// TwinCAT 3 PLC project Clara_20230328
// ProgramVersion: 3.1.4022.7
// CompilerDefines: VISU_USEWSTRING
// libraries:
//   CAA Memory, * (CAA Technical Workgroup)
//   CmpBitmapPool, * (System)
//   Tc2_EtherCAT, * (Beckhoff Automation GmbH)
//   Tc2_IoFunctions, * (Beckhoff Automation GmbH)
//   Tc2_MC2, * (Beckhoff Automation GmbH)
//   Tc2_MDP, * (Beckhoff Automation GmbH)
//   Tc2_ModbusRTU, * (Beckhoff Automation GmbH)
//   Tc2_SerialCom, * (Beckhoff Automation GmbH)
//   Tc2_Standard, * (Beckhoff Automation GmbH)
//   Tc2_SUPS, * (Beckhoff Automation GmbH)
//   Tc2_System, * (Beckhoff Automation GmbH)
//   Tc2_SystemCX, * (Beckhoff Automation GmbH)
//   Tc2_Utilities, * (Beckhoff Automation GmbH)
//   Tc3_Module, * (Beckhoff Automation GmbH)
//   VisuDialogs, * (System)
//   VisuSymbols,3.5.10.0,System
// project tree:
//   DUTs/01_ST_IO/ ST_Input.TcDUT (not stored), ST_IO_FootPedal.TcDUT (not stored), ST_Output.TcDUT
//   DUTs/02_PLC/ stAxis.TcDUT (not stored), stFootPedal.TcDUT, stISS.TcDUT (not stored), stSubTank.TcDUT (not stored), stMaintenanceUnit.TcDUT, stRollToRoll.TcDUT, stRtu.TcDUT (not stored), stSafetyGuard.TcDUT, stSpitUnit.TcDUT (not stored), stSystemEnvironment.TcDUT, stTableVacuum.TcDUT (not stored), stUpDownSlot.TcDUT, stUVLed.TcDUT (not stored)
//   Enum_Text/Enum/PLC/ AxisStateEnum.TcDUT (not stored), Axis_XY_ErrorEnum.TcDUT (not stored), Axis_Z_ErrorEnum.TcDUT, EnvironmentErrorEnum.TcDUT, EnvironmentStateEnum.TcDUT, FootPedalErrorEnum.TcDUT (not stored), FootPedalStateEnum.TcDUT (not stored), ISSErrorEnum.TcDUT (not stored), SubTankErrorEnum.TcDUT, ISSStateEnum.TcDUT, SubTankInkEnum.TcDUT (not stored), SubTankStateEnum.TcDUT (not stored), MUErrorEnum.TcDUT (not stored), MUStateEnum.TcDUT (not stored), RTRErrorEnum.TcDUT, RTRStateEnum.TcDUT, SafetyGuardErrorEnum.TcDUT, SafetyGuardStateEnum.TcDUT, SpitUnitErrorEnum.TcDUT, SpitUnitStateEnum.TcDUT, SwapInfoEnum.TcDUT (not stored), TabVacErrorEnum.TcDUT, TabVacStateEnum.TcDUT (not stored), UpDownSlotErrorEnum.TcDUT, UpDownSlotStateEnum.TcDUT, UVLedErrorEnum.TcDUT, UVLedStateEnum.TcDUT
//   Enum_Text/Enum/TwinSafe/ TwinSAFE_FB_ESTOP_State_Enum.TcDUT (not stored), TwinSAFE_Group_State_Enum.TcDUT
//   Global Variables/ _01_Global_Variables.TcGVL (not stored), _04_Global_Variables_InOutput.TcGVL (not stored)
//   / GlobalTextList.TcGTLO (not stored), ImagePool.TcIPO (not stored), PlcTask.TcTTO (not stored), Task_com.TcTTO (not stored), 视图管理器.TcVMO (not stored)
//   GVLs/ COMM.TcGVL (not stored), GVL.TcGVL (not stored), GVL_Alarm.TcGVL (not stored), GVL_API.TcGVL
//   POUs/000_程序辅助系统/报警/Data types/ Alm_AlarmHistoryType.TcDUT, Alm_AlarmType.TcDUT (not stored), Alm_AlmMsg.TcDUT (not stored), Alm_EventClass.TcDUT (not stored)
//   POUs/000_程序辅助系统/报警/diag_FB/ ethercatinfo_read.TcPOU
//   POUs/000_程序辅助系统/报警/Alarm_FB/ FB_AlarmMain.TcPOU (not stored), FB_DiagDataLogging_S.TcPOU, FB_SetAlarm.TcPOU, SW_FormatWstring.TcPOU (not stored)
//   POUs/000_程序辅助系统/报警/Alarm_FB/Products/ FB_DirectoryCopy.TcPOU, FB_FileCopy.TcPOU (not stored)
//   POUs/000_程序辅助系统/报警/ MAIN_Alarm.TcPOU
//   POUs/000_程序辅助系统/系统功能/ P_UPS.TcPOU, systime.TcPOU (not stored)
//   POUs/001_FB/ FB_Buzzer.TcPOU (not stored), FB_count.TcPOU, FB_SQUARE.TcPOU (not stored), FB_WriteAnalog.TcPOU
//   POUs/002_Modbus/BackPrg/ PRG_COMM.TcPOU (not stored)
//   POUs/002_Modbus/ PRG_SerialComm.TcPOU, P_Modbus.TcPOU (not stored), P_Modbus_RTU.TcPOU
//   POUs/003_Input_Output/ IO_Link.TcPOU (not stored), P_API_IO.TcPOU
//   POUs/010_Motion/MotionBase/ FB_Home_Z.TcPOU, FB_Home_X.TcPOU (not stored), FB_MoveFS_Exte.TcPOU (not stored), FB_MoveSS_Exte.TcPOU (not stored), FB_MoveZ_Exte.TcPOU (not stored)
//   POUs/010_Motion/XMove/ P_FastScan.TcPOU (not stored)
//   POUs/010_Motion/YMove/ P_SlowScan.TcPOU (not stored)
//   POUs/010_Motion/ZMove/ P_Z_Axis.TcPOU (not stored)
//   POUs/030_MediaTransport/TableVacuum/FB/ FB_TableVacuum.TcPOU
//   POUs/030_MediaTransport/UpDownSlot/FB/ FB_UpDownSlotS1.TcPOU (not stored), FB_UpDownSlotS2_S6.TcPOU (not stored)
//   POUs/040_System/FootPedal/FB/ FB_FootPedal.TcPOU (not stored)
//   POUs/040_System/SafetyGuard/FB/ FB_SafetyGuard.TcPOU
//   POUs/040_System/SafetyGuard/ P_SafetyGuard.TcPOU
//   POUs/040_System/SystemEnvironment/FB/ FB_SystemEnvironment.TcPOU (not stored)
//   POUs/050_InkSystem/ISS/ P_ISS.TcPOU (not stored)
//   POUs/050_InkSystem/ P_InkSystem.TcPOU
//   POUs/050_InkSystem/搅拌_吸废墨/FB/ FB_Stirrer.TcPOU
//   POUs/050_InkSystem/搅拌_吸废墨/ P_Stirrer_WastePump.TcPOU
//   POUs/030_MediaTransport/ P_MediaTransport.TcPOU (not stored)
//   POUs/030_MediaTransport/TableVacuum/ P_TableVacuum.TcPOU
//   POUs/030_MediaTransport/UpDownSlot/ P_UpDownSlot.TcPOU
//   POUs/010_Motion/MotionBase/PTP/ Axis_IO.TcPOU (not stored), Axis_PTP_CoE.TcPOU
//   POUs/010_Motion/ P_Motion.TcPOU
//   POUs/060_UVLed/FB/ FB_UVLed_L.TcPOU, FB_UVLed_R.TcPOU
//   POUs/070_RollToRoll/FB/ FB_RollToRoll_Torque.TcPOU (not stored)
//   POUs/100_SubTank/FB/ FB_Circulation.TcPOU (not stored), FB_SubTank_C.TcPOU (not stored), FB_SubTank_W.TcPOU (not stored)
//   POUs/100_SubTank/ P_SubTank.TcPOU
//   POUs/999_TwinSAFE/ P_TwinSAFE.TcPOU (not stored)
//   POUs/ MAIN.TcPOU
//   POUs/070_RollToRoll/ P_RollToRoll.TcPOU
//   POUs/040_System/FootPedal/ P_FootPedal.TcPOU
//   POUs/040_System/ P_System.TcPOU
//   POUs/040_System/SystemEnvironment/ P_SystemEnvironment.TcPOU (not stored)
//   POUs/060_UVLed/ P_UVLed.TcPOU
//   POUs/090MaintenanceUnit/FB/ FB_Auto_Cycles_Swap.TcPOU, FB_drip_purge.TcPOU (not stored)
//   POUs/090MaintenanceUnit/ P_MaintenanceUnit.TcPOU
//   POUs/080SpitUnit/FB/ FB_HomeSpitUnit.TcPOU (not stored), FB_MoveSpitUnit_Exte.TcPOU (not stored)
//   POUs/080SpitUnit/ P_SpitUnit.TcPOU (not stored)
//   VISUs/base/ title.TcVIS (not stored)
//   VISUs/Components/IO_Components/ F99_IO_IO.TcVIS (not stored), F99_IO_IO_1.TcVIS (not stored), F99_IO_IO_2.TcVIS (not stored)
//   VISUs/Components/ VIS_FootPedal.TcVIS, VIS_Drip_purge.TcVIS, VIS_SubTank.TcVIS (not stored), VIS_SystemEnvironment.TcVIS, VIS_ISS.TcVIS, VIS_MU.TcVIS, VIS_RTR_1.TcVIS, VIS_RTR_2.TcVIS (not stored), VIS_SaftyGuard.TcVIS, VIS_SpitUnit.TcVIS (not stored), VIS_TabVac.TcVIS (not stored), VIS_UpDownSlot.TcVIS (not stored)
//   VISUs/HMI_IO监控文字/ EL1809_M_1.TcTLO (not stored), EL1809_M_2.TcTLO (not stored), EL1809_M_3.TcTLO (not stored), EL1809_S_1.TcTLO (not stored), EL1809_S_2.TcTLO, EL1904_M_1.TcTLO (not stored), EL1904_M_2.TcTLO (not stored), EL1904_M_3.TcTLO, EL1904_M_4.TcTLO, EL1904_M_5.TcTLO, EL2809_M_1.TcTLO, EL2809_M_2.TcTLO, EL2809_M_3.TcTLO, EL2809_M_4.TcTLO (not stored), EL2809_S_1.TcTLO, EL2904_M_1.TcTLO
//   VISUs/ F99_Monitor.TcVIS, F7_RTR.TcVIS (not stored), F4_System.TcVIS, F1_AXIS.TcVIS (not stored), F5_InkSystem.TcVIS (not stored), F3_MediaTransport.TcVIS, F6_UVLed.TcVIS
//   VISUs/VIS文本/PLC/ ISS_Object.TcTLO (not stored), subinklevel.TcTLO, TextListSpitUnitErrorid.TcTLO, TextListSpitUnitState.TcTLO (not stored), TextList_EnvironmentError.TcTLO (not stored), TextList_EnvironmentState.TcTLO (not stored), TextList_FootPedalerroid.TcTLO, TextList_SubTankerroid.TcTLO (not stored), TextList_FootPedalstate.TcTLO (not stored), TextList_ISSerrorid.TcTLO (not stored), TextList_ISSstate.TcTLO (not stored), TextList_MU_errorid.TcTLO (not stored), TextList_MU_state.TcTLO (not stored), TextList_RTRstate.TcTLO, TextList_RTR_errorid.TcTLO (not stored), TextList_SafetyGuarderrorid.TcTLO, TextList_SafetyGuardstate.TcTLO (not stored), TextList_SubTank_circuit.TcTLO (not stored), TextList_SwapInfo.TcTLO (not stored), TextList_tabvac_errorid.TcTLO (not stored), TextList_tabvac_state.TcTLO (not stored), TextList_UpDownSlot_errorid.TcTLO (not stored), TextList_UpDownSlot_state.TcTLO (not stored), TextList_UVLed_errorid.TcTLO, TextList_UVLed_state.TcTLO, TextList_xyErrorid.TcTLO (not stored), TextList_xyzState.TcTLO (not stored), TextList_zErrorid.TcTLO
//   VISUs/VIS文本/TwinSafe/ TextList_TwinSAFE_FB_ESTOP_State.TcTLO (not stored), TextList_TwinSAFE_Group_State.TcTLO (not stored)
//   VISUs/报警/ Visualization_ActEvent.TcVIS (not stored), Visualization_LogEvent.TcVIS, vis_arm.TcVIS (not stored)
// real-time tasks:
//   TASK PlcTask: cycle T#10ms, priority 12, ADS port 350
//   TASK Task_com: cycle T#2ms, priority 6, ADS port 352
// motion (NC):
//   TASK NC-Task 1 SAF: cycle T#2ms, priority 4, ADS port 501
//   TASK NC-Task 1 SVB: cycle T#5ms, priority 10, ADS port 511
//   AXIS Axis_FS (id 1)
//     Dynamic: Acceleration=5927.27, Deceleration=5927.27, Jerk=27883
//     Velo: RefSearch=10, RefSync=10, SlowManual=50, FastManual=100
//     TargetPosControl: Time=0.005
//     OtherSettings: AllowMotionCmdToSlave=true
//     encoder EncType=19
//       EncPara: ScaleFactorNumerator=0.001, MaxCount=#xffffffff
//         Inc: RefSearchInverse=true, RefSyncInverse=false
//     drive DrvType=16
//       DrvPara: MaxCount=#xffffffff, DriveControlDWord=#x00020000
//         Analog: VeloReferenz=2000, TorqueSetpointScale=10, ScaleFactorActTorque=0.1
//         TimeComp: TaskDelayCycles=1
//     controller CtrType=1
//       CtrPara: PriorControlFactor=1
//         PosDiffControl: Range=250
//         Observer: BandWidth=20
//   AXIS Axis_SS (id 2)
//     Dynamic: Acceleration=274.92, Deceleration=274.92, Jerk=748.92
//     Velo: Maximum=174
//     OtherSettings: AllowMotionCmdToSlave=true
//     encoder EncType=19
//       EncPara: ScaleFactorNumerator=3.12605035e-07, Inverse=true, MaxCount=#xffffffff
//     drive DrvType=16
//       DrvPara: Inverse=true, MaxCount=#xffffffff, DriveControlDWord=#x00020000
//         Analog: VeloReferenz=180, TorqueSetpointScale=10, ScaleFactorActTorque=0.1
//         TimeComp: TaskDelayCycles=1
//     controller CtrType=1
//       CtrPara: PriorControlFactor=1
//         PosDiffControl: Range=50
//         Observer: BandWidth=20
//   AXIS Z_Axis (id 3)
//     Dynamic: Acceleration=33.4286, Deceleration=33.4286, Jerk=133.032
//     Velo: RefSearch=2, RefSync=2, SlowManual=8, FastManual=10, Maximum=15
//     OtherSettings: AllowMotionCmdToSlave=true
//     encoder EncType=19
//       EncPara: ScaleFactorNumerator=1.7881393e-08, MaxCount=#xffffffff
//         Inc: RefSearchInverse=true, RefSyncInverse=false
//     drive DrvType=16
//       DrvPara: MaxCount=#xffffffff, DriveControlDWord=#x00020000
//         Analog: VeloReferenz=15, TorqueSetpointScale=10, ScaleFactorActTorque=0.1
//         TimeComp: TaskDelayCycles=1
//     controller CtrType=1
//       CtrPara: PriorControlFactor=1
//         PosDiffControl: Range=10
//         Observer: BandWidth=20
//   AXIS Axis_unwider_input1 (id 4)
//     Dynamic: Acceleration=4200, Deceleration=4200, Jerk=14700
//     Velo: SlowManual=60, FastManual=100, Maximum=3000
//     OtherSettings: AllowMotionCmdToSlave=true
//     encoder EncType=19
//       EncPara: ScaleFactorNumerator=3.57628e-06, MaxCount=#xffffffff
//     drive DrvType=16
//       DrvPara: MaxCount=#xffffffff, DriveControlDWord=#x00020000
//         Analog: VeloReferenz=3000, TorqueSetpointScale=10, ScaleFactorActTorque=0.1
//         TimeComp: TaskDelayCycles=1
//     controller CtrType=1
//       CtrPara: PriorControlFactor=1
//         PosDiffControl: Enable=false, Range=100
//         Observer: BandWidth=20
//   AXIS Axis_unwinder_input2 (id 5)
//     Dynamic: Acceleration=4000, Deceleration=4000, Jerk=16000
//     Velo: Maximum=3000
//     OtherSettings: AllowMotionCmdToSlave=true
//     encoder EncType=19
//       EncPara: ScaleFactorNumerator=3.57628e-06, Inverse=true, MaxCount=#xffffffff
//     drive DrvType=16
//       DrvPara: Inverse=true, MaxCount=#xffffffff, DriveControlDWord=#x00020000
//         Analog: VeloReferenz=3000, TorqueSetpointScale=10, ScaleFactorActTorque=0.1
//         TimeComp: TaskDelayCycles=1
//     controller CtrType=1
//       CtrPara: PriorControlFactor=1
//         PosDiffControl: Enable=false, Range=100
//         Observer: BandWidth=20
//   AXIS Axis_winder_output1 (id 6)
//     Dynamic: Acceleration=4000, Deceleration=4000, Jerk=16000
//     Velo: Maximum=3000
//     OtherSettings: AllowMotionCmdToSlave=true
//     encoder EncType=19
//       EncPara: ScaleFactorNumerator=3.57628e-06, MaxCount=#xffffffff
//     drive DrvType=16
//       DrvPara: MaxCount=#xffffffff, DriveControlDWord=#x00020000
//         Analog: VeloReferenz=3000, TorqueSetpointScale=10, ScaleFactorActTorque=0.1
//         TimeComp: TaskDelayCycles=1
//     controller CtrType=1
//       CtrPara: PriorControlFactor=1
//         PosDiffControl: Enable=false, Range=100
//         Observer: BandWidth=20
//   AXIS Axis_winder_output2 (id 7)
//     Dynamic: Acceleration=4000, Deceleration=4000, Jerk=16000
//     Velo: Maximum=3000
//     OtherSettings: AllowMotionCmdToSlave=true
//     encoder EncType=19
//       EncPara: ScaleFactorNumerator=3.57628e-06, Inverse=true, MaxCount=#xffffffff
//     drive DrvType=16
//       DrvPara: Inverse=true, MaxCount=#xffffffff, DriveControlDWord=#x00020000
//         Analog: VeloReferenz=3000, TorqueSetpointScale=10, ScaleFactorActTorque=0.1
//         TimeComp: TaskDelayCycles=1
//     controller CtrType=1
//       CtrPara: PriorControlFactor=1
//         PosDiffControl: Enable=false, Range=100
//         Observer: BandWidth=20
//   AXIS SpitUnit (id 8)
//     Dynamic: Acceleration=32.1429, Deceleration=32.1429, Jerk=137.755
//     Velo: RefSearch=2, RefSync=2, SlowManual=5, FastManual=10, Maximum=15
//     OtherSettings: AllowMotionCmdToSlave=true
//     encoder EncType=19
//       EncPara: ScaleFactorNumerator=1.7881393e-08, Inverse=true, MaxCount=#xffffffff
//         Inc: RefSearchInverse=true, RefSyncInverse=false
//     drive DrvType=16
//       DrvPara: Inverse=true, MaxCount=#xffffffff, DriveControlDWord=#x00020000
//         Analog: VeloReferenz=15, TorqueSetpointScale=10, ScaleFactorActTorque=0.1
//         TimeComp: TaskDelayCycles=1
//     controller CtrType=1
//       CtrPara: PriorControlFactor=1
//         PosDiffControl: Range=10
//         Observer: BandWidth=20
// I/O:
//   DEVICE Device 1 (EtherCAT), AmsNetId 192.168.1.138.2.1
//     Term 1 (EK1200) [EK1200-5000 EtherCAT Power supply (2A E-Bus)]
//       Term 2 (EL1809) [EL1809 16Ch. Dig. Input 24V, 3ms]
//       Term 3 (EL1809) [EL1809 16Ch. Dig. Input 24V, 3ms]
//       Term 4 (EL1809) [EL1809 16Ch. Dig. Input 24V, 3ms]
//       Term 5 (EL2809) [EL2809 16Ch. Dig. Output 24V, 0.5A]
//       Term 6 (EL2809) [EL2809 16Ch. Dig. Output 24V, 0.5A]
//       Term 7 (EL2809) [EL2809 16Ch. Dig. Output 24V, 0.5A]
//       Term 8 (EL6900) [EL6900, TwinSAFE PLC]
//       Term 9 (EL1904) [EL1904, 4 Ch. Safety Input 24V, TwinSAFE]
//         modules: Module 1 (FSOES)
//       Term 10 (EL1904) [EL1904, 4 Ch. Safety Input 24V, TwinSAFE]
//         modules: Module 1 (FSOES)
//       Term 11 (EL1904) [EL1904, 4 Ch. Safety Input 24V, TwinSAFE]
//         modules: Module 1 (FSOES)
//       Term 12 (EL1904) [EL1904, 4 Ch. Safety Input 24V, TwinSAFE]
//         modules: Module 1 (FSOES)
//       Term 13 (EL1904) [EL1904, 4 Ch. Safety Input 24V, TwinSAFE]
//         modules: Module 1 (FSOES)
//       Term 14 (EL9410) [EL9410 E-Bus Power Supplier  (Diagnostics)]
//       Term 15 (EL2904) [EL2904, 4 Ch. Safety Output 24V, 0.5A, TwinSAFE]
//         modules: Module 1 (FSOES), Module 2 (DO)
//       Term 16 (EL2809) [EL2809 16Ch. Dig. Output 24V, 0.5A]
//       Term 17 (EL6001) [EL6001 Interface (RS232)]
//       Term 18 (EL6022) [EL6022 Interface 2Ch. (RS422/485)]
//       Term 19 (EK1110) [EK1110 EtherCAT extension]
//     Drive 20 (ASDA-A3-E CoE Drive) [Delta ASDA-A3-E EtherCAT(CoE) Drive Rev0.05]
//     Drive 21 (ASDA-A3-E CoE Drive) [Delta ASDA-A3-E EtherCAT(CoE) Drive Rev0.05]
//     Drive 22 (ASDA-A3-E CoE Drive) [Delta ASDA-A3-E EtherCAT(CoE) Drive Rev0.05]
//     Drive 23 (ASDA-A3-E CoE Drive) [Delta ASDA-A3-E EtherCAT(CoE) Drive Rev0.05]
//     Drive 24 (ASDA-A3-E CoE Drive) [Delta ASDA-A3-E EtherCAT(CoE) Drive Rev0.05]
//     Drive 25 (ASDA-A3-E CoE Drive) [Delta ASDA-A3-E EtherCAT(CoE) Drive Rev0.05]
//     Drive 26 (ASDA-A3-E CoE Drive) [Delta ASDA-A3-E EtherCAT(CoE) Drive Rev0.05]
//     Drive 27 (ASDA-A3-E CoE Drive) [Delta ASDA-A3-E EtherCAT(CoE) Drive Rev0.05]
//     Term 28 (EK1100) [EK1100 EtherCAT Coupler (2A E-Bus)]
//       Term 29 (EL1809) [EL1809 16Ch. Dig. Input 24V, 3ms]
//       Term 30 (EL1809) [EL1809 16Ch. Dig. Input 24V, 3ms]
//       Term 31 (EL2809) [EL2809 16Ch. Dig. Output 24V, 0.5A]
//       Term 32 (EL4002) [EL4002 2Ch. Ana. Output 0-10V, 12bit]
//       Term 33 (EL9011) [EL9011 End Terminal]
// variable links:
//   Device 1 (EtherCAT) <-> Device 1 (EtherCAT)/Term 1 (EK1200)/Term 10 (EL1904)
//     Term 1 (EK1200)/Term 8 (EL6900)/ConnectionInputs/Message_53 TxPDO <-> Module 1 (FSOES)/RxPDO/FSOE
//   Device 1 (EtherCAT) <-> Device 1 (EtherCAT)/Term 1 (EK1200)/Term 12 (EL1904)
//     Term 1 (EK1200)/Term 8 (EL6900)/ConnectionOutputs/Message_55 RxPDO <-> Module 1 (FSOES)/TxPDO/FSOE
//   Device 1 (EtherCAT) <-> Device 1 (EtherCAT)/Term 1 (EK1200)/Term 13 (EL1904)
//     Term 1 (EK1200)/Term 8 (EL6900)/ConnectionInputs/Message_56 TxPDO <-> Module 1 (FSOES)/RxPDO/FSOE
//     Term 1 (EK1200)/Term 8 (EL6900)/ConnectionOutputs/Message_56 RxPDO <-> Module 1 (FSOES)/TxPDO/FSOE
//   Device 1 (EtherCAT) <-> Device 1 (EtherCAT)/Term 1 (EK1200)/Term 15 (EL2904)
//     Term 1 (EK1200)/Term 8 (EL6900)/ConnectionInputs/Message_57 TxPDO <-> Module 1 (FSOES)/RxPDO/FSOE
//   Device 1 (EtherCAT) <-> Device 1 (EtherCAT)/Term 1 (EK1200)/Term 8 (EL6900)
//     Term 1 (EK1200)/Term 10 (EL1904)/Module 1 (FSOES)/TxPDO/FSOE <-> ConnectionOutputs/Message_53 RxPDO
//     Term 1 (EK1200)/Term 11 (EL1904)/Module 1 (FSOES)/TxPDO/FSOE <-> ConnectionOutputs/Message_58 RxPDO
//     Term 1 (EK1200)/Term 15 (EL2904)/Module 1 (FSOES)/TxPDO/FSOE <-> ConnectionOutputs/Message_57 RxPDO
//     Term 1 (EK1200)/Term 11 (EL1904)/Module 1 (FSOES)/RxPDO/FSOE <-> ConnectionInputs/Message_58 TxPDO
//     Term 1 (EK1200)/Term 12 (EL1904)/Module 1 (FSOES)/RxPDO/FSOE <-> ConnectionInputs/Message_55 TxPDO
//     Term 1 (EK1200)/Term 9 (EL1904)/Module 1 (FSOES)/RxPDO/FSOE <-> ConnectionInputs/Message_52 TxPDO
//   Device 1 (EtherCAT) <-> Device 1 (EtherCAT)/Term 1 (EK1200)/Term 9 (EL1904)
//     Term 1 (EK1200)/Term 8 (EL6900)/ConnectionOutputs/Message_52 RxPDO <-> Module 1 (FSOES)/TxPDO/FSOE
//   NC-Task 1 SAF/Axes/Axis_FS <-> Device 1 (EtherCAT)/Drive 20 (ASDA-A3-E CoE Drive)
//     Drive/Inputs/In/nDataIn3[0] <-> 2nd TxPDO Mapping/Actual Torque
//     Drive/Inputs/In/nDcOutputTime <-> InfoData/DcOutputShift
//     Drive/Inputs/In/nState1 <-> 2nd TxPDO Mapping/Status Word
//     Drive/Inputs/In/nState2 <-> 2nd TxPDO Mapping/Status Word @bit 8
//     Drive/Inputs/In/nState4 @bit 1 <-> WcState/InputToggle
//     Drive/Inputs/In/nState4 <-> WcState/WcState
//     Drive/Outputs/Out/nCtrl1 <-> 2nd RxPDO Mapping/Control Word
//     Drive/Outputs/Out/nCtrl2 <-> 2nd RxPDO Mapping/Control Word @bit 8
//     Drive/Outputs/Out/nDataOut1 <-> 2nd RxPDO Mapping/Target Position
//     Drive/Outputs/Out/nDataOut2 <-> 2nd RxPDO Mapping/Target Velocity
//     Drive/Outputs/Out/nDataOut4[0] <-> 2nd RxPDO Mapping/Target Torque
//     Enc/Inputs/In/nDataIn1 <-> 2nd TxPDO Mapping/Actual Position
//     Enc/Inputs/In/nDataIn3 <-> 2nd TxPDO Mapping/Touch Probe Pos1 Pos Value
//     Enc/Inputs/In/nDataIn7 <-> 2nd TxPDO Mapping/Velocity actual value
//     Enc/Inputs/In/nDcInputTime <-> InfoData/DcInputShift
//     Enc/Inputs/In/nState4 @bit 1 <-> WcState/InputToggle
//     Enc/Inputs/In/nState4 <-> WcState/WcState
//     Enc/Inputs/In/nState5 <-> 2nd TxPDO Mapping/Touch Probe Status
//     Enc/Inputs/In/nState6 <-> 2nd TxPDO Mapping/Touch Probe Status @bit 8
//     Enc/Outputs/Out/nCtrl5 <-> 2nd RxPDO Mapping/Touch Probe Function
//     Enc/Outputs/Out/nCtrl6 <-> 2nd RxPDO Mapping/Touch Probe Function @bit 8
//   NC-Task 1 SAF/Axes/Axis_SS <-> Device 1 (EtherCAT)/Drive 21 (ASDA-A3-E CoE Drive)
//     Drive/Inputs/In/nDataIn3[0] <-> 2nd TxPDO Mapping/Actual Torque
//     Drive/Inputs/In/nDcOutputTime <-> InfoData/DcOutputShift
//     Drive/Inputs/In/nState1 <-> 2nd TxPDO Mapping/Status Word
//     Drive/Inputs/In/nState2 <-> 2nd TxPDO Mapping/Status Word @bit 8
//     Drive/Inputs/In/nState4 @bit 1 <-> WcState/InputToggle
//     Drive/Inputs/In/nState4 <-> WcState/WcState
//     Drive/Outputs/Out/nCtrl1 <-> 2nd RxPDO Mapping/Control Word
//     Drive/Outputs/Out/nCtrl2 <-> 2nd RxPDO Mapping/Control Word @bit 8
//     Drive/Outputs/Out/nDataOut1 <-> 2nd RxPDO Mapping/Target Position
//     Drive/Outputs/Out/nDataOut2 <-> 2nd RxPDO Mapping/Target Velocity
//     Drive/Outputs/Out/nDataOut4[0] <-> 2nd RxPDO Mapping/Target Torque
//     Enc/Inputs/In/nDataIn1 <-> 2nd TxPDO Mapping/Actual Position
//     Enc/Inputs/In/nDataIn3 <-> 2nd TxPDO Mapping/Touch Probe Pos1 Pos Value
//     Enc/Inputs/In/nDataIn7 <-> 2nd TxPDO Mapping/Velocity actual value
//     Enc/Inputs/In/nDcInputTime <-> InfoData/DcInputShift
//     Enc/Inputs/In/nState4 @bit 1 <-> WcState/InputToggle
//     Enc/Inputs/In/nState4 <-> WcState/WcState
//     Enc/Inputs/In/nState5 <-> 2nd TxPDO Mapping/Touch Probe Status
//     Enc/Inputs/In/nState6 <-> 2nd TxPDO Mapping/Touch Probe Status @bit 8
//     Enc/Outputs/Out/nCtrl5 <-> 2nd RxPDO Mapping/Touch Probe Function
//     Enc/Outputs/Out/nCtrl6 <-> 2nd RxPDO Mapping/Touch Probe Function @bit 8
//   NC-Task 1 SAF/Axes/Axis_unwider_input1 <-> Device 1 (EtherCAT)/Drive 23 (ASDA-A3-E CoE Drive)
//     Drive/Inputs/In/nDataIn3[0] <-> 3rd TxPDO Mapping/Actual Torque
//     Drive/Inputs/In/nDcOutputTime <-> InfoData/DcOutputShift
//     Drive/Inputs/In/nState1 <-> 3rd TxPDO Mapping/Status Word
//     Drive/Inputs/In/nState2 <-> 3rd TxPDO Mapping/Status Word @bit 8
//     Drive/Inputs/In/nState4 @bit 1 <-> WcState/InputToggle
//     Drive/Inputs/In/nState4 <-> WcState/WcState
//     Drive/Inputs/In/nState5 <-> 3rd TxPDO Mapping/Mode Of Operation Display
//     Drive/Outputs/Out/nCtrl1 <-> 3rd RxPDO Mapping/Control Word
//     Drive/Outputs/Out/nCtrl2 <-> 3rd RxPDO Mapping/Control Word @bit 8
//     Drive/Outputs/Out/nCtrl5 <-> 3rd RxPDO Mapping/Mode Of Operation
//     Drive/Outputs/Out/nDataOut1 <-> 3rd RxPDO Mapping/Target Position
//     Drive/Outputs/Out/nDataOut2 <-> 3rd RxPDO Mapping/Target Velocity
//     Drive/Outputs/Out/nDataOut4[0] <-> 3rd RxPDO Mapping/Target Torque
//     Enc/Inputs/In/nDataIn1 <-> 3rd TxPDO Mapping/Actual Position
//     Enc/Inputs/In/nDataIn3 <-> 3rd TxPDO Mapping/Touch Probe Pos1 Pos Value
//     Enc/Inputs/In/nDataIn7 <-> 3rd TxPDO Mapping/Velocity actual value
//     Enc/Inputs/In/nDcInputTime <-> InfoData/DcInputShift
//     Enc/Inputs/In/nState4 @bit 1 <-> WcState/InputToggle
//     Enc/Inputs/In/nState4 <-> WcState/WcState
//     Enc/Inputs/In/nState5 <-> 3rd TxPDO Mapping/Touch Probe Status
//     Enc/Inputs/In/nState6 <-> 3rd TxPDO Mapping/Touch Probe Status @bit 8
//     Enc/Outputs/Out/nCtrl5 <-> 3rd RxPDO Mapping/Touch Probe Function
//     Enc/Outputs/Out/nCtrl6 <-> 3rd RxPDO Mapping/Touch Probe Function @bit 8
//   NC-Task 1 SAF/Axes/Axis_unwinder_input2 <-> Device 1 (EtherCAT)/Drive 24 (ASDA-A3-E CoE Drive)
//     Drive/Inputs/In/nDataIn3[0] <-> 3rd TxPDO Mapping/Actual Torque
//     Drive/Inputs/In/nDcOutputTime <-> InfoData/DcOutputShift
//     Drive/Inputs/In/nState1 <-> 3rd TxPDO Mapping/Status Word
//     Drive/Inputs/In/nState2 <-> 3rd TxPDO Mapping/Status Word @bit 8
//     Drive/Inputs/In/nState4 @bit 1 <-> WcState/InputToggle
//     Drive/Inputs/In/nState4 <-> WcState/WcState
//     Drive/Inputs/In/nState5 <-> 3rd TxPDO Mapping/Mode Of Operation Display
//     Drive/Outputs/Out/nCtrl1 <-> 3rd RxPDO Mapping/Control Word
//     Drive/Outputs/Out/nCtrl2 <-> 3rd RxPDO Mapping/Control Word @bit 8
//     Drive/Outputs/Out/nCtrl5 <-> 3rd RxPDO Mapping/Mode Of Operation
//     Drive/Outputs/Out/nDataOut1 <-> 3rd RxPDO Mapping/Target Position
//     Drive/Outputs/Out/nDataOut2 <-> 3rd RxPDO Mapping/Target Velocity
//     Drive/Outputs/Out/nDataOut4[0] <-> 3rd RxPDO Mapping/Target Torque
//     Enc/Inputs/In/nDataIn1 <-> 3rd TxPDO Mapping/Actual Position
//     Enc/Inputs/In/nDataIn3 <-> 3rd TxPDO Mapping/Touch Probe Pos1 Pos Value
//     Enc/Inputs/In/nDataIn7 <-> 3rd TxPDO Mapping/Velocity actual value
//     Enc/Inputs/In/nDcInputTime <-> InfoData/DcInputShift
//     Enc/Inputs/In/nState4 @bit 1 <-> WcState/InputToggle
//     Enc/Inputs/In/nState4 <-> WcState/WcState
//     Enc/Inputs/In/nState5 <-> 3rd TxPDO Mapping/Touch Probe Status
//     Enc/Inputs/In/nState6 <-> 3rd TxPDO Mapping/Touch Probe Status @bit 8
//     Enc/Outputs/Out/nCtrl5 <-> 3rd RxPDO Mapping/Touch Probe Function
//     Enc/Outputs/Out/nCtrl6 <-> 3rd RxPDO Mapping/Touch Probe Function @bit 8
//   NC-Task 1 SAF/Axes/Axis_winder_output1 <-> Device 1 (EtherCAT)/Drive 25 (ASDA-A3-E CoE Drive)
//     Drive/Inputs/In/nDataIn3[0] <-> 3rd Transmit PDO Mapping/Torque actual value
//     Drive/Inputs/In/nDcOutputTime <-> InfoData/DcOutputShift
//     Drive/Inputs/In/nState1 <-> 3rd Transmit PDO Mapping/Statusword
//     Drive/Inputs/In/nState2 <-> 3rd Transmit PDO Mapping/Statusword @bit 8
//     Drive/Inputs/In/nState4 @bit 1 <-> WcState/InputToggle
//     Drive/Inputs/In/nState4 <-> WcState/WcState
//     Drive/Inputs/In/nState5 <-> 3rd Transmit PDO Mapping/Modes of operation display
//     Drive/Outputs/Out/nCtrl1 <-> 3rd Receive PDO Mapping/Controlword
//     Drive/Outputs/Out/nCtrl2 <-> 3rd Receive PDO Mapping/Controlword @bit 8
//     Drive/Outputs/Out/nCtrl5 <-> 3rd Receive PDO Mapping/Modes of operation
//     Drive/Outputs/Out/nDataOut1 <-> 3rd Receive PDO Mapping/Target position
//     Drive/Outputs/Out/nDataOut2 <-> 3rd Receive PDO Mapping/Target velocity
//     Drive/Outputs/Out/nDataOut4[0] <-> 3rd Receive PDO Mapping/Target torque
//     Enc/Inputs/In/nDataIn1 <-> 3rd Transmit PDO Mapping/Position actual value
//     Enc/Inputs/In/nDataIn3 <-> 3rd Transmit PDO Mapping/Touch Probe Pos1 Pos Value
//     Enc/Inputs/In/nDataIn7 <-> 3rd Transmit PDO Mapping/Velocity actual value
//     Enc/Inputs/In/nDcInputTime <-> InfoData/DcInputShift
//     Enc/Inputs/In/nState4 @bit 1 <-> WcState/InputToggle
//     Enc/Inputs/In/nState4 <-> WcState/WcState
//     Enc/Inputs/In/nState5 <-> 3rd Transmit PDO Mapping/Touch Probe Status
//     Enc/Inputs/In/nState6 <-> 3rd Transmit PDO Mapping/Touch Probe Status @bit 8
//     Enc/Outputs/Out/nCtrl5 <-> 3rd Receive PDO Mapping/Touch Probe Function
//     Enc/Outputs/Out/nCtrl6 <-> 3rd Receive PDO Mapping/Touch Probe Function @bit 8
//   NC-Task 1 SAF/Axes/Axis_winder_output2 <-> Device 1 (EtherCAT)/Drive 26 (ASDA-A3-E CoE Drive)
//     Drive/Inputs/In/nDataIn3[0] <-> 3rd TxPDO Mapping/Actual Torque
//     Drive/Inputs/In/nDcOutputTime <-> InfoData/DcOutputShift
//     Drive/Inputs/In/nState1 <-> 3rd TxPDO Mapping/Status Word
//     Drive/Inputs/In/nState2 <-> 3rd TxPDO Mapping/Status Word @bit 8
//     Drive/Inputs/In/nState4 @bit 1 <-> WcState/InputToggle
//     Drive/Inputs/In/nState4 <-> WcState/WcState
//     Drive/Inputs/In/nState5 <-> 3rd TxPDO Mapping/Mode Of Operation Display
//     Drive/Outputs/Out/nCtrl1 <-> 3rd RxPDO Mapping/Control Word
//     Drive/Outputs/Out/nCtrl2 <-> 3rd RxPDO Mapping/Control Word @bit 8
//     Drive/Outputs/Out/nCtrl5 <-> 3rd RxPDO Mapping/Mode Of Operation
//     Drive/Outputs/Out/nDataOut1 <-> 3rd RxPDO Mapping/Target Position
//     Drive/Outputs/Out/nDataOut2 <-> 3rd RxPDO Mapping/Target Velocity
//     Drive/Outputs/Out/nDataOut4[0] <-> 3rd RxPDO Mapping/Target Torque
//     Enc/Inputs/In/nDataIn1 <-> 3rd TxPDO Mapping/Actual Position
//     Enc/Inputs/In/nDataIn3 <-> 3rd TxPDO Mapping/Touch Probe Pos1 Pos Value
//     Enc/Inputs/In/nDataIn7 <-> 3rd TxPDO Mapping/Velocity actual value
//     Enc/Inputs/In/nDcInputTime <-> InfoData/DcInputShift
//     Enc/Inputs/In/nState4 @bit 1 <-> WcState/InputToggle
//     Enc/Inputs/In/nState4 <-> WcState/WcState
//     Enc/Inputs/In/nState5 <-> 3rd TxPDO Mapping/Touch Probe Status
//     Enc/Inputs/In/nState6 <-> 3rd TxPDO Mapping/Touch Probe Status @bit 8
//     Enc/Outputs/Out/nCtrl5 <-> 3rd RxPDO Mapping/Touch Probe Function
//     Enc/Outputs/Out/nCtrl6 <-> 3rd RxPDO Mapping/Touch Probe Function @bit 8
//   NC-Task 1 SAF/Axes/SpitUnit <-> Device 1 (EtherCAT)/Drive 27 (ASDA-A3-E CoE Drive)
//     Drive/Inputs/In/nDataIn3[0] <-> 2nd TxPDO Mapping/Actual Torque
//     Drive/Inputs/In/nDcOutputTime <-> InfoData/DcOutputShift
//     Drive/Inputs/In/nState1 <-> 2nd TxPDO Mapping/Status Word
//     Drive/Inputs/In/nState2 <-> 2nd TxPDO Mapping/Status Word @bit 8
//     Drive/Inputs/In/nState4 @bit 1 <-> WcState/InputToggle
//     Drive/Inputs/In/nState4 <-> WcState/WcState
//     Drive/Outputs/Out/nCtrl1 <-> 2nd RxPDO Mapping/Control Word
//     Drive/Outputs/Out/nCtrl2 <-> 2nd RxPDO Mapping/Control Word @bit 8
//     Drive/Outputs/Out/nDataOut1 <-> 2nd RxPDO Mapping/Target Position
//     Drive/Outputs/Out/nDataOut2 <-> 2nd RxPDO Mapping/Target Velocity
//     Drive/Outputs/Out/nDataOut4[0] <-> 2nd RxPDO Mapping/Target Torque
//     Enc/Inputs/In/nDataIn1 <-> 2nd TxPDO Mapping/Actual Position
//     Enc/Inputs/In/nDataIn3 <-> 2nd TxPDO Mapping/Touch Probe Pos1 Pos Value
//     Enc/Inputs/In/nDataIn7 <-> 2nd TxPDO Mapping/Velocity actual value
//     Enc/Inputs/In/nDcInputTime <-> InfoData/DcInputShift
//     Enc/Inputs/In/nState4 @bit 1 <-> WcState/InputToggle
//     Enc/Inputs/In/nState4 <-> WcState/WcState
//     Enc/Inputs/In/nState5 <-> 2nd TxPDO Mapping/Touch Probe Status
//     Enc/Inputs/In/nState6 <-> 2nd TxPDO Mapping/Touch Probe Status @bit 8
//     Enc/Outputs/Out/nCtrl5 <-> 2nd RxPDO Mapping/Touch Probe Function
//     Enc/Outputs/Out/nCtrl6 <-> 2nd RxPDO Mapping/Touch Probe Function @bit 8
//   NC-Task 1 SAF/Axes/Z_Axis <-> Device 1 (EtherCAT)/Drive 22 (ASDA-A3-E CoE Drive)
//     Drive/Inputs/In/nDataIn3[0] <-> 2nd TxPDO Mapping/Actual Torque
//     Drive/Inputs/In/nDcOutputTime <-> InfoData/DcOutputShift
//     Drive/Inputs/In/nState1 <-> 2nd TxPDO Mapping/Status Word
//     Drive/Inputs/In/nState2 <-> 2nd TxPDO Mapping/Status Word @bit 8
//     Drive/Inputs/In/nState4 @bit 1 <-> WcState/InputToggle
//     Drive/Inputs/In/nState4 <-> WcState/WcState
//     Drive/Outputs/Out/nCtrl1 <-> 2nd RxPDO Mapping/Control Word
//     Drive/Outputs/Out/nCtrl2 <-> 2nd RxPDO Mapping/Control Word @bit 8
//     Drive/Outputs/Out/nDataOut1 <-> 2nd RxPDO Mapping/Target Position
//     Drive/Outputs/Out/nDataOut2 <-> 2nd RxPDO Mapping/Target Velocity
//     Drive/Outputs/Out/nDataOut4[0] <-> 2nd RxPDO Mapping/Target Torque
//     Enc/Inputs/In/nDataIn1 <-> 2nd TxPDO Mapping/Actual Position
//     Enc/Inputs/In/nDataIn3 <-> 2nd TxPDO Mapping/Touch Probe Pos1 Pos Value
//     Enc/Inputs/In/nDataIn7 <-> 2nd TxPDO Mapping/Velocity actual value
//     Enc/Inputs/In/nDcInputTime <-> InfoData/DcInputShift
//     Enc/Inputs/In/nState4 @bit 1 <-> WcState/InputToggle
//     Enc/Inputs/In/nState4 <-> WcState/WcState
//     Enc/Inputs/In/nState5 <-> 2nd TxPDO Mapping/Touch Probe Status
//     Enc/Inputs/In/nState6 <-> 2nd TxPDO Mapping/Touch Probe Status @bit 8
//     Enc/Outputs/Out/nCtrl5 <-> 2nd RxPDO Mapping/Touch Probe Function
//     Enc/Outputs/Out/nCtrl6 <-> 2nd RxPDO Mapping/Touch Probe Function @bit 8
//   Clara_20230328/Clara_20230328 Instance <-> Device 1 (EtherCAT)/Drive 23 (ASDA-A3-E CoE Drive)
//     PlcTask Outputs/P_RollToRoll.Max_profile_velocity[1] <-> 3rd RxPDO Mapping/Max profile velocity
//   Clara_20230328/Clara_20230328 Instance <-> Device 1 (EtherCAT)/Drive 24 (ASDA-A3-E CoE Drive)
//     PlcTask Outputs/P_RollToRoll.Max_profile_velocity[3] <-> 3rd RxPDO Mapping/Max profile velocity
//   Clara_20230328/Clara_20230328 Instance <-> Device 1 (EtherCAT)/Drive 25 (ASDA-A3-E CoE Drive)
//     PlcTask Outputs/P_RollToRoll.Max_profile_velocity[2] <-> 3rd Receive PDO Mapping/Max profile velocity
//   Clara_20230328/Clara_20230328 Instance <-> Device 1 (EtherCAT)/Drive 26 (ASDA-A3-E CoE Drive)
//     PlcTask Outputs/P_RollToRoll.Max_profile_velocity[4] <-> 3rd RxPDO Mapping/Max profile velocity
//   Clara_20230328/Clara_20230328 Instance <-> Device 1 (EtherCAT)/Term 1 (EK1200)/Term 10 (EL1904)
//     PlcTask Inputs/.EL1904_M[2,{1..4}] <-> Module 1 (FSOES)/TxPDO/FSOE/InputChannel{1..4}  (4 links)
//   Clara_20230328/Clara_20230328 Instance <-> Device 1 (EtherCAT)/Term 1 (EK1200)/Term 11 (EL1904)
//     PlcTask Inputs/.EL1904_M[3,{1..4}] <-> Module 1 (FSOES)/TxPDO/FSOE/InputChannel{1..4}  (4 links)
//   Clara_20230328/Clara_20230328 Instance <-> Device 1 (EtherCAT)/Term 1 (EK1200)/Term 12 (EL1904)
//     PlcTask Inputs/.EL1904_M[4,{1..4}] <-> Module 1 (FSOES)/TxPDO/FSOE/InputChannel{1..4}  (4 links)
//   Clara_20230328/Clara_20230328 Instance <-> Device 1 (EtherCAT)/Term 1 (EK1200)/Term 13 (EL1904)
//     PlcTask Inputs/.EL1904_M[5,{1..4}] <-> Module 1 (FSOES)/TxPDO/FSOE/InputChannel{1..4}  (4 links)
//   Clara_20230328/Clara_20230328 Instance <-> Device 1 (EtherCAT)/Term 1 (EK1200)/Term 16 (EL2809)
//     PlcTask Outputs/.EL2809_M[4,{1..16}] <-> Channel {1..16}/Output  (16 links)
//   Clara_20230328/Clara_20230328 Instance <-> Device 1 (EtherCAT)/Term 1 (EK1200)/Term 17 (EL6001)
//     Task_com Inputs/.COMIN2/D[{0..21}] <-> COM Inputs/Data In {0..21}  (22 links)
//     Task_com Inputs/.COMIN2/Status <-> COM Inputs/Status
//     Task_com Outputs/.COMOUT2/Ctrl <-> COM Outputs/Ctrl
//     Task_com Outputs/.COMOUT2/D[{0..21}] <-> COM Outputs/Data Out {0..21}  (22 links)
//   Clara_20230328/Clara_20230328 Instance <-> Device 1 (EtherCAT)/Term 1 (EK1200)/Term 18 (EL6022)
//     PlcTask Inputs/P_Modbus_RTU.master[1].InData/D[{0..21}] <-> COM Inputs Channel 2/Data In {0..21}  (22 links)
//     PlcTask Inputs/P_Modbus_RTU.master[1].InData/Status <-> COM Inputs Channel 2/Status
//     PlcTask Outputs/P_Modbus_RTU.master[1].OutData/Ctrl <-> COM Outputs Channel 2/Ctrl
//     PlcTask Outputs/P_Modbus_RTU.master[1].OutData/D[{0..21}] <-> COM Outputs Channel 2/Data Out {0..21}  (22 links)
//     Task_com Inputs/.COMIN1/D[{0..21}] <-> COM Inputs Channel 1/Data In {0..21}  (22 links)
//     Task_com Inputs/.COMIN1/Status <-> COM Inputs Channel 1/Status
//     Task_com Outputs/.COMOUT1/Ctrl <-> COM Outputs Channel 1/Ctrl
//     Task_com Outputs/.COMOUT1/D[{0..21}] <-> COM Outputs Channel 1/Data Out {0..21}  (22 links)
//   Clara_20230328/Clara_20230328 Instance <-> Device 1 (EtherCAT)/Term 1 (EK1200)/Term 2 (EL1809)
//     PlcTask Inputs/.EL1809_M[1,{1..16}] <-> Channel {1..16}/Input  (16 links)
//   Clara_20230328/Clara_20230328 Instance <-> Device 1 (EtherCAT)/Term 1 (EK1200)/Term 3 (EL1809)
//     PlcTask Inputs/.EL1809_M[2,{1..16}] <-> Channel {1..16}/Input  (16 links)
//   Clara_20230328/Clara_20230328 Instance <-> Device 1 (EtherCAT)/Term 1 (EK1200)/Term 4 (EL1809)
//     PlcTask Inputs/.EL1809_M[3,{1..16}] <-> Channel {1..16}/Input  (16 links)
//   Clara_20230328/Clara_20230328 Instance <-> Device 1 (EtherCAT)/Term 1 (EK1200)/Term 5 (EL2809)
//     PlcTask Outputs/.EL2809_M[1,{1..16}] <-> Channel {1..16}/Output  (16 links)
//   Clara_20230328/Clara_20230328 Instance <-> Device 1 (EtherCAT)/Term 1 (EK1200)/Term 6 (EL2809)
//     PlcTask Outputs/.EL2809_M[2,{1..16}] <-> Channel {1..16}/Output  (16 links)
//   Clara_20230328/Clara_20230328 Instance <-> Device 1 (EtherCAT)/Term 1 (EK1200)/Term 7 (EL2809)
//     PlcTask Outputs/.EL2809_M[3,{1..16}] <-> Channel {1..16}/Output  (16 links)
//   Clara_20230328/Clara_20230328 Instance <-> Device 1 (EtherCAT)/Term 1 (EK1200)/Term 8 (EL6900)
//     PlcTask Inputs/P_TwinSAFE.Com_err <-> StandardInputs/Standard Out Var 46
//     PlcTask Inputs/P_TwinSAFE.FB_err <-> StandardInputs/Standard Out Var 47
//     PlcTask Inputs/P_TwinSAFE.TwinSAFE_Group_State <-> TwinSAFE Group Info Data/TwinSafeGroup1 Info Data/State
//     PlcTask Outputs/P_TwinSAFE.Err_Ack <-> StandardOutputs/Standard In Var 39
//   Clara_20230328/Clara_20230328 Instance <-> Device 1 (EtherCAT)/Term 1 (EK1200)/Term 9 (EL1904)
//     PlcTask Inputs/.EL1904_M[1,{1..4}] <-> Module 1 (FSOES)/TxPDO/FSOE/InputChannel{1..4}  (4 links)
//   Clara_20230328/Clara_20230328 Instance <-> Device 1 (EtherCAT)/Term 28 (EK1100)/Term 29 (EL1809)
//     PlcTask Inputs/.EL1809_S[1,{1..16}] <-> Channel {1..16}/Input  (16 links)
//   Clara_20230328/Clara_20230328 Instance <-> Device 1 (EtherCAT)/Term 28 (EK1100)/Term 30 (EL1809)
//     PlcTask Inputs/.EL1809_S[2,{1..16}] <-> Channel {1..16}/Input  (16 links)
//   Clara_20230328/Clara_20230328 Instance <-> Device 1 (EtherCAT)/Term 28 (EK1100)/Term 31 (EL2809)
//     PlcTask Outputs/.EL2809_S[1,{1..16}] <-> Channel {1..16}/Output  (16 links)
//   Clara_20230328/Clara_20230328 Instance <-> Device 1 (EtherCAT)/Term 28 (EK1100)/Term 32 (EL4002)
//     PlcTask Outputs/.EL4002_S[1] <-> AO Outputs Channel 1/Analog output
//     PlcTask Outputs/.EL4002_S[2] <-> AO Outputs Channel 2/Analog output
//   Clara_20230328/Clara_20230328 Instance <-> NC-Task 1 SAF/Axes/Axis_FS
//     PlcTask Inputs/.Axis[1].Ref.NcToPlc <-> Outputs/ToPlc
//     PlcTask Outputs/.Axis[1].Ref.PlcToNc <-> Inputs/FromPlc
//   Clara_20230328/Clara_20230328 Instance <-> NC-Task 1 SAF/Axes/Axis_SS
//     PlcTask Inputs/.Axis[2].Ref.NcToPlc <-> Outputs/ToPlc
//     PlcTask Outputs/.Axis[2].Ref.PlcToNc <-> Inputs/FromPlc
//   Clara_20230328/Clara_20230328 Instance <-> NC-Task 1 SAF/Axes/Axis_unwider_input1
//     PlcTask Inputs/P_RollToRoll.FB_RoolToRool[1].REF.NcToPlc <-> Outputs/ToPlc
//     PlcTask Outputs/P_RollToRoll.FB_RoolToRool[1].REF.PlcToNc <-> Inputs/FromPlc
//   Clara_20230328/Clara_20230328 Instance <-> NC-Task 1 SAF/Axes/Axis_unwinder_input2
//     PlcTask Inputs/P_RollToRoll.FB_RoolToRool[3].REF.NcToPlc <-> Outputs/ToPlc
//     PlcTask Outputs/P_RollToRoll.FB_RoolToRool[3].REF.PlcToNc <-> Inputs/FromPlc
//   Clara_20230328/Clara_20230328 Instance <-> NC-Task 1 SAF/Axes/Axis_winder_output1
//     PlcTask Inputs/P_RollToRoll.FB_RoolToRool[2].REF.NcToPlc <-> Outputs/ToPlc
//     PlcTask Outputs/P_RollToRoll.FB_RoolToRool[2].REF.PlcToNc <-> Inputs/FromPlc
//   Clara_20230328/Clara_20230328 Instance <-> NC-Task 1 SAF/Axes/Axis_winder_output2
//     PlcTask Inputs/P_RollToRoll.FB_RoolToRool[4].REF.NcToPlc <-> Outputs/ToPlc
//     PlcTask Outputs/P_RollToRoll.FB_RoolToRool[4].REF.PlcToNc <-> Inputs/FromPlc
//   Clara_20230328/Clara_20230328 Instance <-> NC-Task 1 SAF/Axes/SpitUnit
//     PlcTask Inputs/.Axis[4].Ref.NcToPlc <-> Outputs/ToPlc
//     PlcTask Outputs/.Axis[4].Ref.PlcToNc <-> Inputs/FromPlc
//   Clara_20230328/Clara_20230328 Instance <-> NC-Task 1 SAF/Axes/Z_Axis
//     PlcTask Inputs/.Axis[3].Ref.NcToPlc <-> Outputs/ToPlc
//     PlcTask Outputs/.Axis[3].Ref.PlcToNc <-> Inputs/FromPlc

// ---- DUTs/01_ST_IO/ST_Output.TcDUT
TYPE ST_Output :
STRUCT
   
	bqLightGrean            :BOOL;(*绿灯 *)	
 	bqLightYellow			:BOOL;(*黄灯*)	
 	bqLightRed				:BOOL;(*红灯*)	
 	
 (********************ISS********************************)  
	bqStirrerWorkingF		:BOOL;(*正向搅拌*)
	bqStirrerWorkingB		:BOOL;(*负向搅拌*)
	bqWastePump				:BOOL;//吸废墨
	
	bqFillPumpWorking		:ARRAY[1..20] OF BOOL;//
	(*
			墨桶	液位	泵		
1	LC	1,2	1,2	FB_SubInkFeed_C	[1]
2	LM	3,4	3,4	FB_SubInkFeed_C	[2]
3	Y	5,6	5,6	FB_SubInkFeed_C	[3]
4	M	7,8	7,8	FB_SubInkFeed_C	[4]
5	C	9,10	9,10	FB_SubInkFeed_C	[5]
6	K	11,12	11,12	FB_SubInkFeed_C	[6]
7	W	13,14,15,16	13,15	FB_SubInkFeed_W	
8	P	17,18	17,18	FB_SubInkFeed_P	
9	F	19,20	19,20	FB_SubInkFeed_Flush	


	*)
	bqSubCircPumpWorking	:ARRAY[1..2] OF BOOL;	//circulation pump transport the white ink 	
	bqsensor_blink					:ARRAY[1..10] OF BOOL;//
	
	bqPurValve					:BOOL;//V7,正压电磁阀
	bqVacValve_W				:BOOL;//V8,白负压电磁阀
	bqVacValve_C				:BOOL;//V9,彩负压电磁阀

 (********************stSpitUnit********************************)  
	bqFanPower					:BOOL;//废墨吸风
 (********************Z********************************)  	
	bqElectromagnet_power	:BOOL;//探块电源
	
	(****************UpDownSlot********************)
	bqUDS_MoveDown_do		:ARRAY[2..number_UpDownSlot] OF BOOL;		
	bqUDS_MoveUp_do			:ARRAY[2..number_UpDownSlot] OF BOOL;
	bqS1_Drive_enabled				:BOOL;//导向压轮电机使能
	bqS1_Forward_Reverse			:BOOL;//导向压轮电机正/反转
	bqS1_Break							:BOOL;//导向压轮电机刹车
	
	(****************RTR:  1:input1; 2:output1; 3:input2; 4:output2      ********************)
	bqBreakPower           :ARRAY[1..4] OF BOOL;
	bqCluthOut			   :ARRAY[1..4] OF BOOL;
	bqReset				:ARRAY[1..4] OF BOOL;
	
	(****************Table Vacuum********************)
	bqVacRun				:ARRAY[1..number_TableVacuum] OF BOOL;
	(*****************************************)
	bqBuzzer				:BOOL;(*蜂鸣器*)

END_STRUCT
END_TYPE

// ---- DUTs/02_PLC/stFootPedal.TcDUT
TYPE stFootPedal :
STRUCT
//R//
	error_code					:INT;	//	
	state					:INT;	//	
	Error					:BOOL;

//W//
	pressed					:INT;//‘none’, ‘pedal1’, ‘pedal2’, ‘pedal3’
	Reset					:BOOL;
	debounce_time			:LREAL:=500;//ms The amount of time that the foot pedal does not register another click.


	
END_STRUCT
END_TYPE

// ---- DUTs/02_PLC/stMaintenanceUnit.TcDUT
TYPE stMaintenanceUnit :
STRUCT
//R//	
		error_code	:INT;
		state				:INT;
		SwapInfo		:INT;
		has_dripped	:BOOL;	//Indicates if automated dripping was executed at least once after dripping_allowed was enabled
		waste_maximum_level:BOOL;//True if the maximum level in the waste container is reached
		Swapping_Done			:BOOL;
		Error						:BOOL;
		white_circuit_content	:INT;
//W//
	Initialize:BOOL;
	Swap:BOOL;
	cycle:INT;   //"0:Cycle A: Swap white ink to storage ;1:Cycle B: Swap storage to white ink"
	SetOff:BOOL;	
	dripping_allowed:BOOL;   //Indicates if the automated dripping is allowed
	
	IntervalTime_W 			:LREAL;//min
	DripTime_W 				:LREAL;//sec
	PurgeTime_W 			:LREAL;//sec
	IntervalTime_C 			:LREAL;//min
	DripTime_C 				:LREAL;//sec
	PurgeTime_C 			   :LREAL;//sec

END_STRUCT
END_TYPE

// ---- DUTs/02_PLC/stRollToRoll.TcDUT
TYPE stRollToRoll :
STRUCT
//R//
	error_code					:UDINT;	//	
	state					    :INT;	//	
	AxisErrorId					:UDINT;// 轴错误
	initialized					:BOOL;
	error							:BOOL;
	tensioned					:BOOL;
	untensioned				:BOOL;
//W//	
	acceleration				:LREAL:=4200;//	
	deceleration				:LREAL:=4200;//	
	rate						:DINT:=20;//Motor speed or torque.
	untension_rate				:DINT;//Duty cycle for the motor speed during untensioning
	tension_mode				:BOOL;//Indicates the printside: outside	0	The media is loaded outside (cf. following pictures)
	//inside	1	The media is loaded inside (cf. following pictures)
	
	tension_timeout				:LREAL:=2000;//Maximum allowed time for balancer to come in position during ‘tensioning’ state.
	untension_timeout			:LREAL:=2000;//Maximum allowed time to stabilize the system when untensioning the RollToRoll
	brake_timeout				:LREAL:=2000;//the time the brake is allowed to be active. If this is exceeded then an error is set
	Initialize					:BOOL;//
	SetActivate					:BOOL;//
	SetReady					:BOOL;//
	EnableBrake					:BOOL;//
	DisableBrake				:BOOL;//
	StartTension				:BOOL;//
	StopTension					:BOOL;//
	Unlock						:BOOL;//
	Lock						:BOOL;//
	SetOff						:BOOL;//
	is_printing					:BOOL;
	usable			  			:BOOL;
	
END_STRUCT
END_TYPE

// ---- DUTs/02_PLC/stSafetyGuard.TcDUT
TYPE stSafetyGuard :
STRUCT
	//R//
	error_code			:INT;
	state						:INT;
	shuttle_crash_detector_left					:BOOL;
	shuttle_crash_detector_right				:BOOL;
	emergency_stop									:BOOL;
	limit_switch_right								:BOOL;
	limit_switch_left									:BOOL;
	limit_switch_bottom							:BOOL;
	interlock_front_left								:BOOL;
	interlock_front_right							:BOOL;
	interlock_rear_right								:BOOL;
	interlock_rear_left								:BOOL;
	interlock_shuttle_door							:BOOL;
	Interlock_maintenace_door					:BOOL;
	Interlock_spit_door								:BOOL;
	Init_Done											:BOOL;
	Error													:BOOL;

	//W//	
	Initialize			:BOOL;
	SetOff			:BOOL;

	
END_STRUCT
END_TYPE

// ---- DUTs/02_PLC/stSystemEnvironment.TcDUT
TYPE stSystemEnvironment :
STRUCT
//R//
	error_code			:INT;
	state				:INT;
	temp_measured:LREAL;
	humidity_measured:LREAL;
	Error						:BOOL;
//W//	

	Reset:BOOL;
	BuzzerOn:BOOL;
	BuzzerOff:BOOL;
	duration:LREAL;//S
	period :LREAL;//S

	

END_STRUCT
END_TYPE

// ---- DUTs/02_PLC/stUpDownSlot.TcDUT
TYPE stUpDownSlot :
STRUCT
//R//
	error_code				:INT;	//	
	state				:INT;	//		
	sensor_up		    :BOOL;
	sensor_down	        :BOOL;
	Error					:BOOL;
//W//
	Initialize			:BOOL;
	MoveDown			:BOOL;
	MoveUp				:BOOL;
	Setoff				:BOOL;
	timeout_up			:LREAL:=5;//S
	timeout_down		:LREAL:=5;//S
	extra_down_time		:LREAL:=0.1;//S
	

END_STRUCT
END_TYPE

// ---- Enum_Text/Enum/PLC/Axis_Z_ErrorEnum.TcDUT
{attribute 'qualified_only'}
{attribute 'strict'}
{attribute 'to_string'}
TYPE Axis_Z_ErrorEnum :
(
no_error	:=	0	,//	No error detected
not_connected	:=	1	,//	A command was requested prior to opening the driver
invalid_state	:=	2	,//	An invalid command was requested
homing_error	:=	3	,//	The homing sequence failed 
cmd_timeout	:=	4	,//	excute commond timed out
TBD_error	:=	5	,//	
io_error	:=	6	,//	IO error HW board
unknown_error	:=	7	,//	Unknown – Network error
actuator_out_of_pos_range	:=	8	,//	
actuator_out_of_neg_range	:=	9	,//	
homing_timeout	:=	10	,//	
parameter_out_of_range	:=	11	,//	
trigger_Limit	:=	12	,//	limit is triggered
Drive_not_ready_for_operation	:=	13	,//	Drive not ready for operation
interlock_error	:=	14	,
Invalid_IO_data_for_more_than_n_subsequent_NC_cycles_encoder	:=	15	,//	Possible reasons for this error: An EtherCAT slave may have left its OP state or there is a too high real time usage or a too high real time jitter.
				
emergency_error	:=	666	//	



	
);
END_TYPE

// ---- Enum_Text/Enum/PLC/EnvironmentErrorEnum.TcDUT
{attribute 'qualified_only'}
{attribute 'strict'}
{attribute 'to_string'}
TYPE EnvironmentErrorEnum :
(
no_error	:=	0	,//	No error detected
not_connected	:=	1	,//	A command was requested prior to opening the driver
invalid_state	:=	2	,//	An invalid command was requested
io_error	:=	3	,//	IO error HW board
unknown_error	:=	4	,//	Unknown / Network error
emergency_error	:=	666	//	




	
);
END_TYPE

// ---- Enum_Text/Enum/PLC/EnvironmentStateEnum.TcDUT
{attribute 'qualified_only'}
{attribute 'strict'}
{attribute 'to_string'}
TYPE EnvironmentStateEnum :
(
ready	:=	0	,//	The SystemEnvironment is in ready-state.
error	:=	100	//	The SystemEnvironment is in error.



);
END_TYPE

// ---- Enum_Text/Enum/PLC/SubTankErrorEnum.TcDUT
{attribute 'qualified_only'}
{attribute 'strict'}
{attribute 'to_string'}
TYPE SubTankErrorEnum :
(
no_error			:=	0	,//	No error detected
pump_timeout		:=	1	,//	Pump is in error
back_to_air_tank	:=	2	,//	
emergency_error		:=	666	//	

);
END_TYPE

// ---- Enum_Text/Enum/PLC/ISSStateEnum.TcDUT
{attribute 'qualified_only'}
{attribute 'strict'}
{attribute 'to_string'}
TYPE ISSStateEnum :
(
	off	:=	0	,//	The ISS is in off-state.
initializing	:=	1	,//	The ISS is busy initializing.
ready	:=	2	,//	The ISS is ready.
error	:=	100	//	The ISS is in error.


);
END_TYPE

// ---- Enum_Text/Enum/PLC/RTRErrorEnum.TcDUT
{attribute 'qualified_only'}
{attribute 'strict'}
{attribute 'to_string'}
TYPE RTRErrorEnum :
(
no_error	:=	0	,//	No error detected
not_connected	:=	1	,//	A command was requested prior to opening the driver
invalid_state	:=	2	,//	An invalid command was requested
break_exceeded_timeout	:=	3	,//	
cmd_timeout	:=	4	,//	excute commond timed out
unknown_error	:=	5	,//	Unknown – Network error
Drive_not_ready_for_operation	:=	6	,//	Drive not ready for operation
roll_unclamped	:=	7	,//
Invalid_IO_data_for_more_than_n_subsequent_NC_cycles_encoder	:=	8	,//	Possible reasons for this error: An EtherCAT slave may have left its OP state or there is a too high real time usage or a too high real time jitter.

emergency_error	:=	666	//	The object is in error due to an active emergency error.



);
END_TYPE

// ---- Enum_Text/Enum/PLC/RTRStateEnum.TcDUT
{attribute 'qualified_only'}
{attribute 'strict'}
{attribute 'to_string'}
TYPE RTRStateEnum :
(
off	:=	0	,//	The RollToRoll object is switched off
initializing	:=	1	,//	The RollToRoll is busy initializing
ready	:=	2	,//	The RollToRoll is ready to use
active	:=	4	,//	The RollToRoll is active
tensioning	:=	5	,//	The RollToRoll is busy tensioning
Tensioned_locked	:=	6	,//	The RollToRoll is tensioned
tensioned	:=	8	,//	The RollToRoll is tensioned
untensioning	:=	9	,//	The RollToRoll is busy untensioning
setting_off	:=	10	,//	"The RollToRoll is going to off. If needed it is busy untensioning for off.All errors - except emergency stop error - will be ignored."
brake_enabled	:=	13	,//	The RollToRoll is locked
error	:=	100	//	The RollToRoll is in error


);
END_TYPE

// ---- Enum_Text/Enum/PLC/SafetyGuardErrorEnum.TcDUT
{attribute 'qualified_only'}
{attribute 'strict'}
{attribute 'to_string'}
TYPE SafetyGuardErrorEnum :
(
no_error	:=	0	,//	No error detected
not_connected	:=	1	,//	A command was requested prior to opening the driver
invalid_state	:=	2	,//	An invalid command was requested
emergency_error	:=	4	,//	Emergency error
interlock_error	:=	8	,//	Interlock error
shuttle_crash_error	:=	16	,//	Shuttle crash error
limit_switch_error	:=	32	,//	Limit switch error
io_error	:=	64	,//	IO error HW board
unknown_error	:=	128	//	Unknown / Network error


);
END_TYPE

// ---- Enum_Text/Enum/PLC/SafetyGuardStateEnum.TcDUT
{attribute 'qualified_only'}
{attribute 'strict'}
{attribute 'to_string'}
TYPE SafetyGuardStateEnum :
(
off	:=	0	,//	The SafetyGuard is off
initializing	:=	1	,//	The SafetyGuard is busy initializing
ready	:=	2	,//	The SafetyGuard is in ready-state.
error	:=	100	//	The SafetyGuard is in error.


);
END_TYPE

// ---- Enum_Text/Enum/PLC/SpitUnitErrorEnum.TcDUT
{attribute 'qualified_only'}
{attribute 'strict'}
{attribute 'to_string'}
TYPE SpitUnitErrorEnum :
(
no_error	:=	0	,//	No error detected
not_connected	:=	1	,//	A command was requested prior to opening the driver
invalid_state	:=	2	,//	An invalid command was requested
homing_error	:=	3	,//	When the homing position cannot be detected, the moving distance may not exceed the specified maxDistance parameter
trigger_limit	:=	4	,//
io_error	:=	5	,//
unknown_error	:=	6	,//
Drive_not_ready_for_operation	:=	7	,//	Drive not ready for operation
Invalid_IO_data_for_more_than_n_subsequent_NC_cycles_encoder	:=	8	,//	Possible reasons for this error: An EtherCAT slave may have left its OP state or there is a too high real time usage or a too high real time jitter.
parameter_out_of_range	:=	9	,//

emergency_error	:=	666	//


);
END_TYPE

// ---- Enum_Text/Enum/PLC/SpitUnitStateEnum.TcDUT
{attribute 'qualified_only'}
{attribute 'strict'}
{attribute 'to_string'}
TYPE SpitUnitStateEnum :
(
off	:=	0	,//	The SpitUnit is in off-state.
initializing	:=	1	,//	The SpitUnit is busy initializing.
homing	:=	2	,//	The Home command started successful. The SpitUnit is moving
ready	:=	3	,//	The Home command finished successful and the SpitUnit is idle again. Or The Move command finished successful and the SpitUnit is idle again
moving	:=	4	,//	The Move command started successful. The SpitUnit is moving
error	:=	100	//	The SpitUnit is in error.

);
END_TYPE

// ---- Enum_Text/Enum/PLC/TabVacErrorEnum.TcDUT
{attribute 'qualified_only'}
{attribute 'strict'}
{attribute 'to_string'}

TYPE TabVacErrorEnum :
(
no_error	:=	0	,//	No error detected
not_connected	:=	1	,//	A command was requested prior to opening the driver
invalid_state	:=	2	,//	An invalid command was requested
vacuum_on_timeout	:=	3	,//	
vacuum_off_timeout	:=	4	,//	
cmd_timeout	:=	5	,//	
TBD_error	:=	6	,//	
io_error	:=	7	,//	IO error HW board
unknown_error	:=	8	,//	Unknown – Network error
emergency_error	:=	666	//	


);
END_TYPE

// ---- Enum_Text/Enum/PLC/UpDownSlotErrorEnum.TcDUT
{attribute 'qualified_only'}
{attribute 'strict'}
{attribute 'to_string'}
TYPE UpDownSlotErrorEnum :
(
no_error	:=	0	,//	No error detected
not_connected	:=	1	,//	A command was requested prior to opening the driver
invalid_state	:=	2	,//	An invalid command was requested
timeout_up	:=	3	,//	Timeout. The UpDownSlot isn’t up left
timeout_down	:=	4	,//	Timeout. The UpDownSlot isn’t down left
cmd_timeout	:=	5	,//	excute commond timed out
io_error	:=	6	,//	IO error HW board
unknown_error	:=	7	,//	Unknown – Network error
emergency_error	:=	666	//	



);
END_TYPE

// ---- Enum_Text/Enum/PLC/UpDownSlotStateEnum.TcDUT
{attribute 'qualified_only'}
{attribute 'strict'}
{attribute 'to_string'}
TYPE UpDownSlotStateEnum :
(
	
	off				:=	0	,//	The UpDownSlot is in off-state.
	up				:=	1	,//	The UpDownSlot is in the upper-position.
	down			:=	2	,//	The UpDownSlot is in the lower-position.
	waiting_up		:=	4	,//	The UpDownSlot object is waiting until the upper position is reached.
	waiting_down	:=	5	,//	The UpDownSlot object is waiting until the lower position is reached
	error			:=	100	//	The UpDownSlot is in error.

);
END_TYPE

// ---- Enum_Text/Enum/PLC/UVLedErrorEnum.TcDUT
{attribute 'qualified_only'}
{attribute 'strict'}
{attribute 'to_string'}
TYPE UVLedErrorEnum :
(
no_error		:=	0	,//	No error detected
not_connected	:=	1	,//	A command was requested prior to opening the driver
invalid_state	:=	2	,//	An invalid command was requested
unknown_error	:=	3,	//Unknown – Network error
abnormal_temperature	:=	4	,//	indicates abnormal temperature

emergency_error:=666//The object is in error due to an active emergency error.

);
END_TYPE

// ---- Enum_Text/Enum/PLC/UVLedStateEnum.TcDUT
{attribute 'qualified_only'}
{attribute 'strict'}
{attribute 'to_string'}
TYPE UVLedStateEnum :
(
	off					:=	0	,//	The UVLed is in off-state.
	initializing		:=	1	,//	The UVLed is busy initializing.
	ready				:=	2	,//	The UVLed is in ready.
	applying_settings	:=	3	,//	"The UVLed is configuring with the curing setting at the start of the print.The UVLed has stopped curing (LEDs are off), as the FS encoder value is leaving the curing window. Settings are re-applied during the end of the swath, preparing the next swath."
	settings_applied	:=	4	,//	The UVLed has finished configuring the power settings.
	ready_for_curing	:=	10	,//	The UVLed is configured with the positions where to cure.The UVLed is ready for curing.
	curing				:=	5	,//	The UVLed is started with curing (LEDs are on), as the FS encoder value is entering the curing window.
	setting_off			:=	6	,//	The UVLed is going to off. If needed LEDs are first cooling down before set in off.
	error				:=	100	//	The UVLed is in error.

);
END_TYPE

// ---- Enum_Text/Enum/TwinSafe/TwinSAFE_Group_State_Enum.TcDUT
{attribute 'qualified_only'}
{attribute 'strict'}
{attribute 'to_string'}
TYPE TwinSAFE_Group_State_Enum :
(
RUN	:=	1	,(*	"Input RUN=1, no error in the group, and all connections have started
up without error"	*)
STOP	:=	2	,(*	Input RUN = 0	*)
ERROR	:=	4	,(*	Group is in error, see Diagnostic information	*)
RESET	:=	5	,(*	"After a group error has occurred, all errors have been rectified and the
Err Ack signal is 1"	*)
START	:=	6	,(*	"The group remains in this state as long as not all connections have
started up after the start of the group (RUN=1)"	*)
STOPERROR	:=	7	,(*	"When the group is started or initialized, it assumes the STOPERROR
status if the TwinSAFE connections are assigned to the group.
The group switches from STOPERROR state into ERROR state if the
Run input is TRUE."	*)
DEACTIVE	:=	16	,(*	Group was deactivated via customizing	*)
WAITCOMERROR	:=	17	(*	"This state is set when the customizing function ""Passivate"" is selected
and the system waits for ComError of the group"	*)

);
END_TYPE

// ---- POUs/000_程序辅助系统/报警/Data types/Alm_AlarmHistoryType.TcDUT
TYPE Alm_AlarmHistoryType :
STRUCT
  	EventMessage:            	WSTRING(255);
	EventId:					DINT;
   	EventTime:               	DT;
END_STRUCT
END_TYPE

// ---- GVLs/GVL_API.TcGVL
{attribute 'qualified_only'}
VAR_GLOBAL
(***************************AXIS*****************************************)	
		stAxis      	     :ARRAY[1..3] OF stAxis;           //伺服轴    
	
(***************************Ink System*****************************************)
	    stISS					:ARRAY[1..9] OF stISS;//LC,LM,Y,M,C,K,W,P,F
		stMU					:stMaintenanceUnit;
		
(***************************TableVacuum*****************************************)
		stTableVacuum    :ARRAY[1..number_TableVacuum] OF stTableVacuum ;	

(***************************UpDownSlot*****************************************)	
		stUpDownSlot	  :ARRAY [1..number_UpDownSlot] OF stUpDownSlot;				//S1-S6		
		
(***************************SYSTEM*****************************************)		
				(***************************FootPedal**************************)	
					stFootPedal		  :ARRAY[1..number_FootPedal] OF stFootPedal;
				(***************************SystemEnvironment**************************)	
					stSystemEnvironment		:stSystemEnvironment;
(***************************UVLed*****************************************)			
		stUVLed			  :ARRAY[1..2] OF stUVLed;
			
(***************************Unw/Rew*****************************************)		
		stRoolToRool	  :ARRAY[1..number_RoolToRool] OF stRollToRoll;//1:input1; 2:output1; 3:input2; 4:output2
		
(***************************InkVacuum*****************************************)
	//R//
		cInkVacCur	:LREAL;//彩墨负压实际值
		wInkVacCur	:LREAL;//白墨负压实际值
	//W//
		cInkVacSet	:LREAL;//彩墨负压设定
		wInkVacSet	:LREAL;//白墨负压设定
	
(***************************UV*****************************************)
	//W//
		UVpowerL		:LREAL;		//0-10V,UV功率
		UVpowerR		:LREAL;		//0-10V,UV功率
		UVlightL		:BOOL;		//UV快门
		UVlightR    	:BOOL;		//UV快门

(***************************SpitUnit *****************************************)		
		stSpitUnit   :stSpitUnit;
		
(***************************SAFE*****************************************)
	//R//
		stSafetyGuard	:stSafetyGuard;
		
(***************************LED*****************************************)
		LEDPower		:BOOL;		//LED灯
(***************************count*****************************************)
		count			:INT;
		Docan			:BOOL;
(***************************SubTank*****************************************)
		stSubTank		:ARRAY[1..16] OF stSubTank;
		
(*****************************************************************)
		stInput					:ST_Input;
		stOutput				:ST_Output;
		Axis_SpitUnit_snHome    :BOOL;
		Axis_SpitUnit_snLimitP  :BOOL;

END_VAR

// ---- POUs/000_程序辅助系统/报警/diag_FB/ethercatinfo_read.TcPOU
FUNCTION_BLOCK ethercatinfo_read
VAR_INPUT
	netID AT %I*:Tc2_System.T_AmsNetIdArr;							//硬件网络的AMSnetID
	nEcMasterDeviceId AT %I*:UINT;											//主站的deviceID
END_VAR
VAR_OUTPUT
	slaveAddresses    : ARRAY[0..255] OF UINT;						//读取的从站地址（以数组保存）
	devStates           : ARRAY[0..255] OF ST_EcSlaveState;		//读取的从站状态机
	slavenames			: ARRAY[0..255] OF T_MaxString;			//读取从站名字
    color					: ARRAY[0..255] OF DWORD;					//显示图标的颜色
	nSlaves           : UINT := 0;														//从站个数
END_VAR
VAR
	i:INT;
	i1:INT;
	NAN:Tc2_System.T_MaxString;											//复位变量
	ton1:Tc2_Standard.TON;														//读取时钟触发器
	bExecute          :  BOOL;															//触发位
	fb_getalladdr:Tc2_EtherCAT.FB_EcGetAllSlaveAddr;		//读取从站地址的功能块 https://infosys.beckhoff.com/content/1033/tcplclib_tc2_ethercat/9007199311752331.html?id=8671424095593379685
	fb_getallstate:Tc2_EtherCAT.FB_EcGetAllSlaveStates;		//读取从站状态机的功能块 https://infosys.beckhoff.com/content/1033/tcplclib_tc2_ethercat/9007199311770635.html?id=2217456128990928132
	fb_getallname: IOF_GetBoxNameByAddr;							//读取从站名称 https://infosys.beckhoff.com/content/1033/tcplclib_tc2_iofunctions/9007199313832971.html?id=4102389766817989774
END_VAR

ton1(IN:= NOT ton1.Q, PT:= T#0.5S, Q=> bExecute, ET=> );

fb_getalladdr(//读取从站地址
	sNetId:= F_CreateAmsNetId(netID), //网络netID
	pAddrBuf:= ADR(slaveAddresses), //寄存器地址
	cbBufLen:= SIZEOF(slaveAddresses), 
	bExecute:= bExecute, 
	nSlaves=> nSlaves);//从站个数
	
fb_getallstate(//读取从站状态机
	sNetId:= F_CreateAmsNetId(netID), //网络地址
	pStateBuf:= ADR(devStates), //寄存器地址
	cbBufLen:= SIZEOF(devStates), 
	bExecute:= bExecute, 
	nSlaves=> );

fb_getallname(//读取从站名称
	NETID:= , 
	DEVICEID:=nEcMasterDeviceId, //device number
	BOXADDR:=  slaveAddresses[i], //从站号
	BOXNAME=> slavenames[i]);//返回从站名

IF slaveAddresses[i]>0 AND NOT fb_getallname .start THEN//反复触发功能块
	fb_getallname.START:=TRUE;
ELSIF slaveAddresses[i+1]>0 AND NOT fb_getallname.BUSY THEN
		i:=i+1;
		fb_getallname.START:=FALSE;
END_IF

FOR i1:=0 TO  nSlaves BY 1 DO//颜色变量触发逻辑
CASE devStates [i1].deviceState OF
	1: color[i1]:=16#FFFF0000;
	2: color[i1]:=16#FFFFFF00;
	4: color[i1]:=16#FF88FF00;
	8: color[i1]:=16#FF00FF00;
	ELSE
	color[i1]:=16#FFFFFFFF;
END_CASE
END_FOR

END_FUNCTION_BLOCK

// ---- POUs/000_程序辅助系统/报警/Alarm_FB/FB_DiagDataLogging_S.TcPOU
FUNCTION_BLOCK FB_DiagDataLogging_S
(*历史文件夹操作*)
VAR_INPUT
	bInUse:							BOOL:=TRUE;(*是否使能功能*)
	bCopyToUSB:						BOOL;(*把文件夹复制到u盘*)

	b_DiagDataLog_AutoDelete:		BOOL:=TRUE;	(* Auto Deletion of Logged Files / highly recommended!	*)(*是否自动删除文件*)
	n_DiagDataLog_KeepForWeeks:		INT:=4;

	bDiagDataLogRunOn_WinCE:		BOOL:=FALSE;
	cnst_DiagDataLogFilePath_XP:	STRING(255):='C:\';
	cnst_DiagDataLogFilePath_CE:	STRING(255):='Hard Disk\';

	cnst_USB_FilePath_XP:			STRING(255):='E:\';
	cnst_USB_FilePath_CE:			STRING(255):='Hard Disk2\';

	cnst_SubDir_DiagDataLog:		STRING(255):='DiagDataLog\';(*文件夹名称*)
	cnst_FileName:					STRING(255):='Sym';(*文件的前缀名*)

END_VAR
VAR_IN_OUT
	sInputString:					STRING(255);(*请先转换成utf8的格式*)
END_VAR
VAR_OUTPUT
	bBusyWriting:					BOOL;
	sWriteData:						STRING(255);
END_VAR
VAR
	nTaskIdx:						BYTE:=0;
	fbGetTaskIdx:					GETCURTASKINDEX;
	fCycleTime:						LREAL;//s

	StartUp:						BOOL:=TRUE;
	count:							INT;
	dtemp:							DINT;
	dtemp2:							DINT;
	stemp:							STRING(255);
	stemp_Del:						STRING(255);
	btemp:							BOOL;

	aStringBuffer:					ARRAY[1..10] OF STRING(255);
	sActUseingString:				STRING(255);
	bInputDoWrite:					BOOL;

	nWrState:						INT;
	sWrite:							STRING(255);
	stWrTime:						TIMESTRUCT;
	fbFormat:						FB_FormatString;
	fbOpen:							FB_FileOpen;
	fbWrite:						FB_FileWrite;
	fbClose:						FB_FileClose;

	nState:							INT;
	nEntries:						INT;
	fbMakeDir:						FB_CreateDir;
	fbGetTime:						NT_GetTime;
	msecond:						UDINT;

	delstep:						INT:=0;
	CopyStep: 						INT:=0;
	deldatestart:					TIMESTRUCT;
	deldate:						TIMESTRUCT;
	fbdelete:						FB_FileDelete;
	fbDirectoryCopy:				FB_DirectoryCopy;
	fdeltime:						LREAL;
	ntemp:							INT;// save days
	sFile:							STRING(255);
	bClearLined:					BOOL;

	bInitialWrite:					BOOL:=TRUE;
	bFirstLog:						BOOL:=TRUE;

	bDiagDataLog_Release : 			BOOL;
	stDiagDataLogTime:				TIMESTRUCT;

	i: INT;
	by_day_or_hour				:BOOL;//1:by_day,0:by_hour
END_VAR

IF NOT bInUse THEN(*是否使能功能*)
	StartUp:=TRUE;
	RETURN;
END_IF

IF StartUp THEN
	(* get cycle time of this task	*)
	fbGetTaskIdx();
	nTaskIdx:=MAX(MIN(fbGetTaskIdx.index,4),1);
	fCycleTime:=UDINT_TO_LREAL(_TaskInfo[nTaskIdx].CycleTime)/10000000.0;
	nState:=0;
	IF fCycleTime<>0 THEN
		StartUp:=FALSE;
	END_IF
END_IF

act_CheckCom();		(*命令处理*)
//act_Copy2USB();		(*复制到其它文件夹*)
IF by_day_or_hour  THEN 	
	act_AutoWrite_by_day();
	act_AutoDelete_by_day();
ELSE
	act_AutoWrite_by_hour();	(*写*)
	act_AutoDelete_by_hour();	(*删除旧文件*)
END_IF

ACTION act_AutoDelete_by_day:

CASE delstep OF
0://获取删除开始时间
	fdeltime:=10.0;
	IF b_DiagDataLog_AutoDelete AND (stDiagDataLogTime.wYear>0) AND (n_DiagDataLog_KeepForWeeks>0) THEN
		ntemp:=1+7*MIN(MAX(n_DiagDataLog_KeepForWeeks,4),4000);//计算保存days+1
		deldate:=stDiagDataLogTime;//
		WHILE (ntemp>0) DO
			IF (deldate.wDay<2) THEN
				deldate.wDay:=deldate.wDay+28;
				deldate.wMonth:=deldate.wMonth-1;
				IF (deldate.wMonth<1) THEN
					deldate.wMonth:=12;
					deldate.wYear:=deldate.wYear-1;
				END_IF
			END_IF
			IF (deldate.wDay=ntemp) THEN//假如相等，表明在单月，从1号开始算
				deldate.wDay:=1;
				ntemp:=1;
			ELSIF (deldate.wDay>ntemp) THEN
				deldate.wDay:=deldate.wDay-ntemp;
				ntemp:=0;
			ELSE
				ntemp:=ntemp-deldate.wDay;
				deldate.wDay:=1;
			END_IF
		END_WHILE
		deldatestart:=deldate;
		delstep:=1;
	END_IF

1:	//第一次10S跳步骤2，下一次每1.5S跳一次
	fdeltime:=fdeltime-fCycleTime;
	IF NOT b_DiagDataLog_AutoDelete THEN
		delstep:=0;
	ELSIF (fdeltime<=0.0) THEN
		delstep:=2;
	END_IF

2://根据删除时间，生成删除文件名，并进行删除
	IF bDiagDataLogRunOn_WinCE THEN
		sFile:=CONCAT(cnst_DiagDataLogFilePath_CE,cnst_SubDir_DiagDataLog);
	ELSE
		sFile:=CONCAT(cnst_DiagDataLogFilePath_XP,cnst_SubDir_DiagDataLog);
	END_IF
	sFile:=CONCAT(sFile,cnst_FileName);
	stemp_Del:=WORD_TO_STRING(deldate.wYear);
	stemp_Del:=CONCAT(stemp_Del,'_');
	IF (deldate.wMonth<10) THEN
		stemp_Del:=CONCAT(stemp_Del,'0');
	END_IF
	stemp_Del:=CONCAT(stemp_Del,WORD_TO_STRING(deldate.wMonth));
	stemp_Del:=CONCAT(stemp_Del,'_');
	IF (deldate.wDay<10) THEN
		stemp_Del:=CONCAT(stemp_Del,'0');
	END_IF
	stemp_Del:=CONCAT(stemp_Del,WORD_TO_STRING(deldate.wDay));
	(*stemp_Del:=CONCAT(stemp_Del,'_');
	IF(deldate.wHour<10)THEN
		stemp_Del:=CONCAT(stemp_Del,'0');
	END_IF
	stemp_Del:=CONCAT(stemp_Del,WORD_TO_STRING(deldate.wHour));
	*)
	stemp_Del:=CONCAT(stemp_Del,'.LOG');
	fbdelete.sPathName:=CONCAT(sFile,stemp_Del);
	fbdelete.bExecute:=TRUE;
	delstep:=3;

3://生成下一个删除时间，每过24个月重新回到1，记录开始删除时间
	IF NOT fbdelete.bBusy THEN
		fbdelete.bExecute:=FALSE;
		(*IF (deldate.wHour=0) THEN
			deldate.wHour:=23;
			deldate.wDay:=deldate.wDay-1;
		ELSE
			deldate.wHour:=deldate.wHour-1;
		END_IF*)
		deldate.wDay:=deldate.wDay-1;
		IF (deldate.wDay<1) THEN
			deldate.wDay:=31;
			deldate.wMonth:=deldate.wMonth-1;
		END_IF
		IF (deldate.wMonth<1) THEN
			deldate.wMonth:=12;
			deldate.wYear:=deldate.wYear-1;
		END_IF
		fdeltime:=1.5;
		dtemp:=12*WORD_TO_DINT(deldatestart.wYear-deldate.wYear)+WORD_TO_DINT(deldatestart.wMonth-deldate.wMonth);//已删除的月数
		IF (dtemp>24) THEN//删除月数大于24个月，重新开始
			delstep:=0;
		ELSE
			delstep:=1;
		END_IF
	END_IF

ELSE
	delstep:=0;

END_CASE

fbdelete();
END_ACTION

ACTION act_AutoDelete_by_hour:

CASE delstep OF
0://获取删除开始时间
	fdeltime:=10.0;
	IF b_DiagDataLog_AutoDelete AND (stDiagDataLogTime.wYear>0) AND (n_DiagDataLog_KeepForWeeks>0) THEN
		ntemp:=1+7*MIN(MAX(n_DiagDataLog_KeepForWeeks,4),4000);//计算保存days+1
		deldate:=stDiagDataLogTime;//
		WHILE (ntemp>0) DO
			IF (deldate.wDay<2) THEN
				deldate.wDay:=deldate.wDay+28;
				deldate.wMonth:=deldate.wMonth-1;
				IF (deldate.wMonth<1) THEN
					deldate.wMonth:=12;
					deldate.wYear:=deldate.wYear-1;
				END_IF
			END_IF
			IF (deldate.wDay=ntemp) THEN//假如相等，表明在单月，从1号开始算
				deldate.wDay:=1;
				ntemp:=1;
			ELSIF (deldate.wDay>ntemp) THEN
				deldate.wDay:=deldate.wDay-ntemp;
				ntemp:=0;
			ELSE
				ntemp:=ntemp-deldate.wDay;
				deldate.wDay:=1;
			END_IF
		END_WHILE
		deldatestart:=deldate;
		delstep:=1;
	END_IF

1:	//第一次10S跳步骤2，下一次每1.5S跳一次
	fdeltime:=fdeltime-fCycleTime;
	IF NOT b_DiagDataLog_AutoDelete THEN
		delstep:=0;
	ELSIF (fdeltime<=0.0) THEN
		delstep:=2;
	END_IF

2://根据删除时间，生成删除文件名，并进行删除
	IF bDiagDataLogRunOn_WinCE THEN
		sFile:=CONCAT(cnst_DiagDataLogFilePath_CE,cnst_SubDir_DiagDataLog);
	ELSE
		sFile:=CONCAT(cnst_DiagDataLogFilePath_XP,cnst_SubDir_DiagDataLog);
	END_IF
	sFile:=CONCAT(sFile,cnst_FileName);
	stemp_Del:=WORD_TO_STRING(deldate.wYear);
	stemp_Del:=CONCAT(stemp_Del,'_');
	IF (deldate.wMonth<10) THEN
		stemp_Del:=CONCAT(stemp_Del,'0');
	END_IF
	stemp_Del:=CONCAT(stemp_Del,WORD_TO_STRING(deldate.wMonth));
	stemp_Del:=CONCAT(stemp_Del,'_');
	IF (deldate.wDay<10) THEN
		stemp_Del:=CONCAT(stemp_Del,'0');
	END_IF
	stemp_Del:=CONCAT(stemp_Del,WORD_TO_STRING(deldate.wDay));
	stemp_Del:=CONCAT(stemp_Del,'_');
	IF(deldate.wHour<10)THEN
		stemp_Del:=CONCAT(stemp_Del,'0');
	END_IF
	stemp_Del:=CONCAT(stemp_Del,WORD_TO_STRING(deldate.wHour));
	stemp_Del:=CONCAT(stemp_Del,'.LOG');
	fbdelete.sPathName:=CONCAT(sFile,stemp_Del);
	fbdelete.bExecute:=TRUE;
	delstep:=3;

3://生成下一个删除时间，每过24个月重新回到1，记录开始删除时间
	IF NOT fbdelete.bBusy THEN
		fbdelete.bExecute:=FALSE;
		IF (deldate.wHour=0) THEN
			deldate.wHour:=23;
			deldate.wDay:=deldate.wDay-1;
		ELSE
			deldate.wHour:=deldate.wHour-1;
		END_IF
		IF (deldate.wDay<1) THEN
			deldate.wDay:=31;
			deldate.wMonth:=deldate.wMonth-1;
		END_IF
		IF (deldate.wMonth<1) THEN
			deldate.wMonth:=12;
			deldate.wYear:=deldate.wYear-1;
		END_IF
		fdeltime:=1.5;
		dtemp:=12*WORD_TO_DINT(deldatestart.wYear-deldate.wYear)+WORD_TO_DINT(deldatestart.wMonth-deldate.wMonth);//已删除的月数
		IF (dtemp>24) THEN//删除月数大于24个月，重新开始
			delstep:=0;
		ELSE
			delstep:=1;
		END_IF
	END_IF

ELSE
	delstep:=0;

END_CASE

fbdelete();
END_ACTION

ACTION act_AutoWrite_by_day:
(*以“年月日时”为名称。也就是说，每小时产生一个
新的文件，以防止文件过大
*)

CASE nState OF

0:	(*wait for clearance*)
	nEntries:=0;
	bInputDoWrite:=bDiagDataLog_Release:=FALSE;
	nWrState:=0;
	IF NOT StartUp THEN
		nState:=1;
	END_IF

1:	(*try to create the directory*)
	fbMakeDir.bExecute:=FALSE;
	fbGetTime.START:=FALSE;
	fbMakeDir.sNetId:='';
	IF bDiagDataLogRunOn_WinCE THEN
		fbMakeDir.sPathName:=CONCAT(cnst_DiagDataLogFilePath_CE,cnst_SubDir_DiagDataLog);
	ELSE
		fbMakeDir.sPathName:=CONCAT(cnst_DiagDataLogFilePath_XP,cnst_SubDir_DiagDataLog);
	END_IF
	fbMakeDir.ePath:=PATH_GENERIC;
	fbMakeDir.tTimeout:=T#5s;
	nState:=2;

2:	fbMakeDir();
	fbGetTime();
	IF NOT fbMakeDir.bExecute THEN
		fbMakeDir.bExecute:=TRUE;
	ELSIF NOT fbMakeDir.bBusy THEN
		IF NOT fbGetTime.START THEN
			fbGetTime.START:=TRUE;
		ELSIF NOT fbGetTime.BUSY THEN
			IF fbGetTime.ERR THEN
				stDiagDataLogTime.wYear:=stDiagDataLogTime.wMonth:=stDiagDataLogTime.wDay:=0;
				stDiagDataLogTime.wHour:=stDiagDataLogTime.wMinute:=stDiagDataLogTime.wSecond:=0;
				stDiagDataLogTime.wMilliseconds:=0;
				msecond:=0;
			ELSE
				stDiagDataLogTime:=fbGetTime.TIMESTR;
				msecond:=fbGetTime.TIMESTR.wMilliseconds;
			END_IF
			fbGetTime(START:=FALSE);
			fbMakeDir(bExecute:=FALSE);
			nState:=11;
		END_IF
	END_IF


11:
	IF(nState>=10)THEN
		(*update and/or synchronize the clock*)
		stDiagDataLogTime.wMilliseconds:=stDiagDataLogTime.wMilliseconds+LREAL_TO_WORD(MIN(MAX(1000.0*fCycleTime,1.0),30000.0));
	
		IF(stDiagDataLogTime.wMilliseconds>=1000)THEN
			stDiagDataLogTime.wMilliseconds:=stDiagDataLogTime.wMilliseconds-1000;
			stDiagDataLogTime.wSecond:=stDiagDataLogTime.wSecond+1;
			IF(stDiagDataLogTime.wSecond>=60)THEN
				stDiagDataLogTime.wSecond:=stDiagDataLogTime.wSecond-60;
				stDiagDataLogTime.wMinute:=stDiagDataLogTime.wMinute+1;
				IF(stDiagDataLogTime.wMinute>=60)THEN
					stDiagDataLogTime.wMinute:=stDiagDataLogTime.wMinute-60;
					stDiagDataLogTime.wHour:=stDiagDataLogTime.wHour+1;
				END_IF
			END_IF
		END_IF
		msecond:=msecond+LREAL_TO_WORD(MIN(MAX(1000.0*fCycleTime,1.0),30000.0));
		fbGetTime(START:=(msecond>1100));
		IF fbGetTime.START THEN
			IF(NOT fbGetTime.BUSY)THEN
				IF(fbGetTime.ERR)THEN
					msecond:=0;
				ELSE
					stDiagDataLogTime:=fbGetTime.TIMESTR;
					msecond:=fbGetTime.TIMESTR.wMilliseconds;
				END_IF
			END_IF
		END_IF

		CASE nWrState OF

			0:	IF bInputDoWrite THEN
					bBusyWriting:= TRUE;
					IF bDiagDataLogRunOn_WinCE THEN
						sWrite:=CONCAT(cnst_DiagDataLogFilePath_CE,cnst_SubDir_DiagDataLog);
					ELSE
						sWrite:=CONCAT(cnst_DiagDataLogFilePath_XP,cnst_SubDir_DiagDataLog);//C:\DiagDataLog\
					END_IF
					sWrite:=CONCAT(sWrite,cnst_FileName);//C:\DiagDataLog\Sym
					stWrTime:=stDiagDataLogTime;
					stemp:=WORD_TO_STRING(stWrTime.wYear);//2020
					stemp:=CONCAT(stemp,'_');////2020_
					IF(stWrTime.wMonth<10)THEN//月份小于10，在月前加0
						stemp:=CONCAT(stemp,'0');////2020_06
					END_IF
					stemp:=CONCAT(stemp,WORD_TO_STRING(stWrTime.wMonth));
					stemp:=CONCAT(stemp,'_');//2020_06_
					IF(stWrTime.wDay<10)THEN
						stemp:=CONCAT(stemp,'0');
					END_IF
					stemp:=CONCAT(stemp,WORD_TO_STRING(stWrTime.wDay));//2020_06_30
					(*stemp:=CONCAT(stemp,'_');//2020_06_30_
					IF(stWrTime.wHour<10)THEN
						stemp:=CONCAT(stemp,'0');
					END_IF
					stemp:=CONCAT(stemp,WORD_TO_STRING(stWrTime.wHour));//2020_06_30_14,把小时记录
					*)
					stemp:=CONCAT(stemp,'.LOG');//2020_06_30_14.LOG,把小时记录
					fbOpen.sPathName:=CONCAT(sWrite,stemp);//C:\DiagDataLog\2020_06_30_14.LOG,完整名称
					fbOpen.bExecute:=FALSE;
					nWrState:=1;
				END_IF
	
			1:	fbOpen(sNetId:='', nMode:=FOPEN_MODEAPPEND OR FOPEN_MODETEXT, ePath:=PATH_GENERIC, tTimeout:=T#5S);
				IF NOT fbOpen.bExecute THEN
					fbOpen.bExecute:=TRUE;
				ELSIF NOT fbOpen.bBusy THEN
					IF fbOpen.bError THEN
						bInputDoWrite:=FALSE;
						nWrState:=0;
					ELSE
						fbWrite(sNetId:='', hFile:=fbOpen.hFile, pWriteBuff:=0, cbWriteLen:=0, bExecute:=FALSE, tTimeout:=T#5s);
						fbClose(sNetId:='', hFile:=fbOpen.hFile, bExecute:=FALSE, tTimeout:=T#5s);
						nWrState:=2;
					END_IF
					fbOpen(bExecute:=FALSE);
				END_IF

			2:	(**)
					stemp:=WORD_TO_STRING(stWrTime.wYear);
					stemp:=CONCAT(stemp,'.');
					IF(stWrTime.wMonth<10)THEN
						stemp:=CONCAT(stemp,'0');
					END_IF
					stemp:=CONCAT(stemp,WORD_TO_STRING(stWrTime.wMonth));
					stemp:=CONCAT(stemp,'.');
					IF(stWrTime.wDay<10)THEN
						stemp:=CONCAT(stemp,'0');
					END_IF
					stemp:=CONCAT(stemp,WORD_TO_STRING(stWrTime.wDay));
					stemp:=CONCAT(stemp,'|');
					IF(stWrTime.wHour<10)THEN
						stemp:=CONCAT(stemp,'0');
					END_IF
					stemp:=CONCAT(stemp,WORD_TO_STRING(stWrTime.wHour));
					stemp:=CONCAT(stemp,':');
					IF(stWrTime.wMinute<10)THEN
						stemp:=CONCAT(stemp,'0');
					END_IF
					stemp:=CONCAT(stemp,WORD_TO_STRING(stWrTime.wMinute));
					stemp:=CONCAT(stemp,':');
					IF(stWrTime.wSecond<10)THEN
						stemp:=CONCAT(stemp,'0');
					END_IF
					stemp:=CONCAT(stemp,WORD_TO_STRING(stWrTime.wSecond));
					stemp:=CONCAT(stemp,':');
					IF(stWrTime.wMilliseconds<10)THEN
						stemp:=CONCAT(stemp,'00');
					END_IF
					IF(stWrTime.wMilliseconds<100)
					AND stWrTime.wMilliseconds>=10 THEN
						stemp:=CONCAT(stemp,'0');
					END_IF
					stemp:=CONCAT(stemp,WORD_TO_STRING(stWrTime.wMilliseconds));
					stemp:=CONCAT(stemp,'|');
					string_to_utf8(ADR(sTemp),ADR(STemp),SIZEOF(sTemp));//强制转换成utf8的格式，才能显示中文

				sWriteData:=sWrite:=CONCAT((stemp) , sActUseingString);
				sWrite:=CONCAT(sWrite,'$n');
				fbWrite(pWriteBuff:=ADR(sWrite), cbWriteLen:=LEN(sWrite), bExecute:=TRUE);
				nWrState:=3;

			3:	fbWrite(pWriteBuff:=ADR(sWrite), cbWriteLen:=LEN(sWrite), bExecute:=TRUE);
				IF NOT fbWrite.bBusy THEN
					IF fbWrite.bError THEN
						nWrState:=-4;
					ELSE
						nWrState:=10;
					END_IF
					fbWrite(bExecute:=FALSE);
				END_IF

			-4,
			10:fbClose(bExecute:=TRUE);
				IF NOT fbClose.bBusy THEN
					IF fbClose.bError THEN
						bBusyWriting:=FALSE;
						bInputDoWrite:=FALSE;
						nWrState:=0;
					ELSE
						bBusyWriting:=FALSE;
						bInputDoWrite:=FALSE;
						nWrState:=0;
					END_IF
					fbClose(bExecute:=FALSE);
				END_IF
		END_CASE
	END_IF



END_CASE
END_ACTION

ACTION act_AutoWrite_by_hour:
(*以“年月日时”为名称。也就是说，每小时产生一个
新的文件，以防止文件过大
*)

CASE nState OF

0:	(*wait for clearance*)
	nEntries:=0;
	bInputDoWrite:=bDiagDataLog_Release:=FALSE;
	nWrState:=0;
	IF NOT StartUp THEN
		nState:=1;
	END_IF

1:	(*try to create the directory*)
	fbMakeDir.bExecute:=FALSE;
	fbGetTime.START:=FALSE;
	fbMakeDir.sNetId:='';
	IF bDiagDataLogRunOn_WinCE THEN
		fbMakeDir.sPathName:=CONCAT(cnst_DiagDataLogFilePath_CE,cnst_SubDir_DiagDataLog);
	ELSE
		fbMakeDir.sPathName:=CONCAT(cnst_DiagDataLogFilePath_XP,cnst_SubDir_DiagDataLog);
	END_IF
	fbMakeDir.ePath:=PATH_GENERIC;
	fbMakeDir.tTimeout:=T#5s;
	nState:=2;

2:	fbMakeDir();
	fbGetTime();
	IF NOT fbMakeDir.bExecute THEN
		fbMakeDir.bExecute:=TRUE;
	ELSIF NOT fbMakeDir.bBusy THEN
		IF NOT fbGetTime.START THEN
			fbGetTime.START:=TRUE;
		ELSIF NOT fbGetTime.BUSY THEN
			IF fbGetTime.ERR THEN
				stDiagDataLogTime.wYear:=stDiagDataLogTime.wMonth:=stDiagDataLogTime.wDay:=0;
				stDiagDataLogTime.wHour:=stDiagDataLogTime.wMinute:=stDiagDataLogTime.wSecond:=0;
				stDiagDataLogTime.wMilliseconds:=0;
				msecond:=0;
			ELSE
				stDiagDataLogTime:=fbGetTime.TIMESTR;
				msecond:=fbGetTime.TIMESTR.wMilliseconds;
			END_IF
			fbGetTime(START:=FALSE);
			fbMakeDir(bExecute:=FALSE);
			nState:=11;
		END_IF
	END_IF


11:
	IF(nState>=10)THEN
		(*update and/or synchronize the clock*)
		stDiagDataLogTime.wMilliseconds:=stDiagDataLogTime.wMilliseconds+LREAL_TO_WORD(MIN(MAX(1000.0*fCycleTime,1.0),30000.0));
	
		IF(stDiagDataLogTime.wMilliseconds>=1000)THEN
			stDiagDataLogTime.wMilliseconds:=stDiagDataLogTime.wMilliseconds-1000;
			stDiagDataLogTime.wSecond:=stDiagDataLogTime.wSecond+1;
			IF(stDiagDataLogTime.wSecond>=60)THEN
				stDiagDataLogTime.wSecond:=stDiagDataLogTime.wSecond-60;
				stDiagDataLogTime.wMinute:=stDiagDataLogTime.wMinute+1;
				IF(stDiagDataLogTime.wMinute>=60)THEN
					stDiagDataLogTime.wMinute:=stDiagDataLogTime.wMinute-60;
					stDiagDataLogTime.wHour:=stDiagDataLogTime.wHour+1;
				END_IF
			END_IF
		END_IF
		msecond:=msecond+LREAL_TO_WORD(MIN(MAX(1000.0*fCycleTime,1.0),30000.0));
		fbGetTime(START:=(msecond>1100));
		IF fbGetTime.START THEN
			IF(NOT fbGetTime.BUSY)THEN
				IF(fbGetTime.ERR)THEN
					msecond:=0;
				ELSE
					stDiagDataLogTime:=fbGetTime.TIMESTR;
					msecond:=fbGetTime.TIMESTR.wMilliseconds;
				END_IF
			END_IF
		END_IF

		CASE nWrState OF

			0:	IF bInputDoWrite THEN
					bBusyWriting:= TRUE;
					IF bDiagDataLogRunOn_WinCE THEN
						sWrite:=CONCAT(cnst_DiagDataLogFilePath_CE,cnst_SubDir_DiagDataLog);
					ELSE
						sWrite:=CONCAT(cnst_DiagDataLogFilePath_XP,cnst_SubDir_DiagDataLog);//C:\DiagDataLog\
					END_IF
					sWrite:=CONCAT(sWrite,cnst_FileName);//C:\DiagDataLog\Sym
					stWrTime:=stDiagDataLogTime;
					stemp:=WORD_TO_STRING(stWrTime.wYear);//2020
					stemp:=CONCAT(stemp,'_');////2020_
					IF(stWrTime.wMonth<10)THEN//月份小于10，在月前加0
						stemp:=CONCAT(stemp,'0');////2020_06
					END_IF
					stemp:=CONCAT(stemp,WORD_TO_STRING(stWrTime.wMonth));
					stemp:=CONCAT(stemp,'_');//2020_06_
					IF(stWrTime.wDay<10)THEN
						stemp:=CONCAT(stemp,'0');
					END_IF
					stemp:=CONCAT(stemp,WORD_TO_STRING(stWrTime.wDay));//2020_06_30
					stemp:=CONCAT(stemp,'_');//2020_06_30_
					IF(stWrTime.wHour<10)THEN
						stemp:=CONCAT(stemp,'0');
					END_IF
					stemp:=CONCAT(stemp,WORD_TO_STRING(stWrTime.wHour));//2020_06_30_14,把小时记录
					stemp:=CONCAT(stemp,'.LOG');//2020_06_30_14.LOG,把小时记录
					fbOpen.sPathName:=CONCAT(sWrite,stemp);//C:\DiagDataLog\2020_06_30_14.LOG,完整名称
					fbOpen.bExecute:=FALSE;
					nWrState:=1;
				END_IF
	
			1:	fbOpen(sNetId:='', nMode:=FOPEN_MODEAPPEND OR FOPEN_MODETEXT, ePath:=PATH_GENERIC, tTimeout:=T#5S);
				IF NOT fbOpen.bExecute THEN
					fbOpen.bExecute:=TRUE;
				ELSIF NOT fbOpen.bBusy THEN
					IF fbOpen.bError THEN
						bInputDoWrite:=FALSE;
						nWrState:=0;
					ELSE
						fbWrite(sNetId:='', hFile:=fbOpen.hFile, pWriteBuff:=0, cbWriteLen:=0, bExecute:=FALSE, tTimeout:=T#5s);
						fbClose(sNetId:='', hFile:=fbOpen.hFile, bExecute:=FALSE, tTimeout:=T#5s);
						nWrState:=2;
					END_IF
					fbOpen(bExecute:=FALSE);
				END_IF

			2:	(**)
					stemp:=WORD_TO_STRING(stWrTime.wYear);
					stemp:=CONCAT(stemp,'.');
					IF(stWrTime.wMonth<10)THEN
						stemp:=CONCAT(stemp,'0');
					END_IF
					stemp:=CONCAT(stemp,WORD_TO_STRING(stWrTime.wMonth));
					stemp:=CONCAT(stemp,'.');
					IF(stWrTime.wDay<10)THEN
						stemp:=CONCAT(stemp,'0');
					END_IF
					stemp:=CONCAT(stemp,WORD_TO_STRING(stWrTime.wDay));
					stemp:=CONCAT(stemp,'|');
					IF(stWrTime.wHour<10)THEN
						stemp:=CONCAT(stemp,'0');
					END_IF
					stemp:=CONCAT(stemp,WORD_TO_STRING(stWrTime.wHour));
					stemp:=CONCAT(stemp,':');
					IF(stWrTime.wMinute<10)THEN
						stemp:=CONCAT(stemp,'0');
					END_IF
					stemp:=CONCAT(stemp,WORD_TO_STRING(stWrTime.wMinute));
					stemp:=CONCAT(stemp,':');
					IF(stWrTime.wSecond<10)THEN
						stemp:=CONCAT(stemp,'0');
					END_IF
					stemp:=CONCAT(stemp,WORD_TO_STRING(stWrTime.wSecond));
					stemp:=CONCAT(stemp,':');
					IF(stWrTime.wMilliseconds<10)THEN
						stemp:=CONCAT(stemp,'00');
					END_IF
					IF(stWrTime.wMilliseconds<100)
					AND stWrTime.wMilliseconds>=10 THEN
						stemp:=CONCAT(stemp,'0');
					END_IF
					stemp:=CONCAT(stemp,WORD_TO_STRING(stWrTime.wMilliseconds));
					stemp:=CONCAT(stemp,'|');
					string_to_utf8(ADR(sTemp),ADR(STemp),SIZEOF(sTemp));//强制转换成utf8的格式，才能显示中文

				sWriteData:=sWrite:=CONCAT((stemp) , sActUseingString);
				sWrite:=CONCAT(sWrite,'$n');
				fbWrite(pWriteBuff:=ADR(sWrite), cbWriteLen:=LEN(sWrite), bExecute:=TRUE);
				nWrState:=3;

			3:	fbWrite(pWriteBuff:=ADR(sWrite), cbWriteLen:=LEN(sWrite), bExecute:=TRUE);
				IF NOT fbWrite.bBusy THEN
					IF fbWrite.bError THEN
						nWrState:=-4;
					ELSE
						nWrState:=10;
					END_IF
					fbWrite(bExecute:=FALSE);
				END_IF

			-4,
			10:fbClose(bExecute:=TRUE);
				IF NOT fbClose.bBusy THEN
					IF fbClose.bError THEN
						bBusyWriting:=FALSE;
						bInputDoWrite:=FALSE;
						nWrState:=0;
					ELSE
						bBusyWriting:=FALSE;
						bInputDoWrite:=FALSE;
						nWrState:=0;
					END_IF
					fbClose(bExecute:=FALSE);
				END_IF
		END_CASE
	END_IF



END_CASE
END_ACTION

ACTION act_CheckCom:
	IF sInputString<>'' AND nState=11 THEN
		FOR i:=1 TO 10 DO
			IF aStringBuffer[i]='' THEN
				aStringBuffer[i]:=sInputString;
				EXIT;
			END_IF
		END_FOR
		sInputString:='';
	END_IF

	IF aStringBuffer[1]<>''AND NOT bInputDoWrite THEN
		sActUseingString:=aStringBuffer[1];
		FOR i:=1 TO 9 DO
			aStringBuffer[i]:= aStringBuffer[i+1];
		END_FOR
		aStringBuffer[10]:='';
		bInputDoWrite:=TRUE;
	END_IF
END_ACTION

ACTION act_Copy2USB:
CASE CopyStep OF
	0:
		IF bCopyToUSB THEN
			CopyStep:=100;
		END_IF

	100:
		IF bDiagDataLogRunOn_WinCE THEN
			fbDirectoryCopy.srcPathName:=cnst_DiagDataLogFilePath_CE;
			fbDirectoryCopy.destPathName:=cnst_USB_FilePath_CE;
		ELSE
			fbDirectoryCopy.srcPathName:=cnst_DiagDataLogFilePath_XP;
			fbDirectoryCopy.destPathName:=cnst_USB_FilePath_XP;
		END_IF
		fbDirectoryCopy.DirectoryName:= LEFT(cnst_SubDir_DiagDataLog,LEN(cnst_SubDir_DiagDataLog)-1);
		fbDirectoryCopy.FileType:= 		'log';
		CopyStep:=200;

	200:
		fbDirectoryCopy(bExecute:=TRUE);
		IF fbDirectoryCopy.bBusy THEN
			CopyStep:=300;
		END_IF

	300:
		fbDirectoryCopy();
		IF NOT fbDirectoryCopy.bBusy THEN
			fbDirectoryCopy(bExecute:=FALSE);
			CopyStep:=400;
		END_IF

	400:
		IF NOT bCopyToUSB THEN
			CopyStep:=0;
		END_IF

END_CASE
END_ACTION

END_FUNCTION_BLOCK

// ---- POUs/000_程序辅助系统/报警/Alarm_FB/Products/FB_DirectoryCopy.TcPOU
(**************最终使用的文件复制功能块*********************)
FUNCTION_BLOCK FB_DirectoryCopy
VAR_INPUT
	srcNetId				: T_AmsNetId;	(* TwinCAT network address of the source file *)
	srcPathName			: T_MaxString;	(* source file path *)(*源的地址*)
	destNetId			: T_AmsNetId;	(* TwinCAT network address of the destination file *)
	destPathName		: T_MaxString;  	(* destination file path  *)(*目标的上层地址*)
	DirectoryName		: T_MaxString;  	(* destination file  name *)(*目标文件夹名字*)
	FileType				: STRING:='*';  		(* destination file  name *)(*文件类型*)
	bExecute			: BOOL;			(* rising edge start fb execution *)
	bFindFileList			: BOOL;			(* rising edge start fb execution *)
	tAdsTimeOut			: TIME;			(* ads timeout *)
	bContinueWhenErr	:BOOL;
	bCancelWhenErr		:BOOL;
END_VAR
VAR_OUTPUT
	bBusy				:BOOL;
	bError				:BOOL;
	nErrId				:UDINT;
	(*==============
	ErrId:=1;		(*ErrId: no find source dir*)
	ErrId:=2;		(*ErrId: no find target dir*)
	ErrId:=3:		target have same file;
	ErrId:=4:		(*Input parameter error*)
	================*)
END_VAR
VAR
	Step				:DWORD;
	RisingEdge			:R_TRIG;
	fbFindFileList:			FB_EnumFindFileList;
	fbEnumFindFileEntry:	FB_EnumFindFileEntry;
	srcFilesLists:			 ARRAY[1..12]  OF ST_FindFileEntry;
	destFilesLists:		 ARRAY[1..12]  OF ST_FindFileEntry;
	fbFileCopy:			FB_FileCopy;
	fbCreateDir:			FB_CreateDir;
	i: 					INT;
	n:					INT;
	bFindFileListState		: BOOL;
	TimeCount:			 INT;
END_VAR

RisingEdge(CLK:=bExecute OR bFindFileList);

IF bBusy THEN
	TimeCount:=TimeCount+1;
END_IF

CASE Step OF
	0:	(* do nothing *)
		IF RisingEdge.Q  AND NOT bBusy THEN
			IF bFindFileList THEN
				bFindFileListState:=TRUE;
				bBusy := TRUE;
				Step := 40;
			ELSE
				bFindFileListState:=FALSE;
				IF DirectoryName=''
				OR FileType=''
				OR srcPathName=''
				OR destPathName='' THEN		(*Input parameter error*)
					bError:=TRUE;
					nErrId:=4;
				ELSE
					bBusy := TRUE;
					bError:= FALSE;
					TimeCount:=0;
					nErrId:=0;
					Step := 10;
				END_IF
			END_IF
		END_IF

	10:	(* find source dir*)
		fbEnumFindFileEntry
			(
			sNetId:='' , 
			sPathName:=CONCAT(srcPathName,DirectoryName),
			eCmd:=eEnumCmd_First ,
			bExecute:=TRUE ,
			tTimeout:=T#10s ,
			);
		IF NOT  fbEnumFindFileEntry.bBusy THEN
			IF NOT  fbEnumFindFileEntry.bEOE THEN		(*target dir is exist*)
				Step := 20;
			ELSE										(*target dir no exist*)
				bError:=TRUE;
				nErrId:=1;		(*ErrId: no find source dir*)
				Step:=70;
			END_IF
			fbEnumFindFileEntry(bExecute:=FALSE);
		END_IF

	11:	(*Wait*)
		IF bContinueWhenErr OR bCancelWhenErr THEN
			bError:=FALSE;
			nErrId:=0;
			Step:=0;
		END_IF

	20:	(*find Target Dir*)
		fbEnumFindFileEntry
			(
			sNetId:='' , 
			sPathName:=CONCAT(destPathName,DirectoryName),
			eCmd:=eEnumCmd_First ,
			bExecute:=TRUE ,
			tTimeout:=T#10s ,
			);
		IF NOT  fbEnumFindFileEntry.bBusy THEN
			IF NOT  fbEnumFindFileEntry.bEOE THEN	(*target dir is exist*)
				Step := 40;
			ELSE									(*target dir no exist*)
				Step:=30;
			END_IF
			fbEnumFindFileEntry(bExecute:=FALSE);
		END_IF

	30:	(*createt dir  *)
		fbCreateDir
			(
			sNetId:='',
			sPathName:= CONCAT(destPathName,DirectoryName),
			ePath:= PATH_GENERIC,
			bExecute:=TRUE,
			tTimeout:=t#10s
			);
		IF NOT fbCreateDir.bBusy THEN
			fbCreateDir(bExecute:=FALSE);
			Step:=40;
		END_IF

	40:	(*Find source FileList*)
		fbFindFileList
			(
			sNetID:='',
			sPathName:=CONCAT(CONCAT(CONCAT(srcPathName,DirectoryName),'\*.'),FileType),
			eCmd:= eEnumCmd_First,
			pFindList:= ADR(srcFilesLists),
			cbFindList:=SIZEOF(srcFilesLists),
			bExecute:= TRUE ,
			tTimeout:=t#10s
			);
		IF NOT fbFindFileList.bBusy THEN
			fbFindFileList(bExecute:=FALSE);
			IF bFindFileList OR bFindFileListState THEN
				Step:=70;
			ELSE
				Step:=41;
			END_IF
		END_IF

	41:	(*Find target FileList*)
		fbFindFileList
			(
			sNetID:='',
			sPathName:=CONCAT(CONCAT(CONCAT(destPathName,DirectoryName),'\*.'),FileType),
			eCmd:= eEnumCmd_First,
			pFindList:= ADR(destFilesLists),
			cbFindList:=SIZEOF(destFilesLists),
			bExecute:= TRUE ,
			tTimeout:=t#10s
			);
		IF NOT fbFindFileList.bBusy THEN
			fbFindFileList(bExecute:=FALSE);
			Step:=50;
			i:=1;
		END_IF


	50:	(*check no same mane file*)
		IF srcFilesLists[i].sFileName='' THEN
			IF i>=15 THEN
				i:=1;
				Step:=70;
			ELSE
				i:=i+1;
			END_IF
		ELSE
			FOR n:=1 TO 15 DO
				IF destFilesLists[n].sFileName =  srcFilesLists[i].sFileName THEN
					bError:=TRUE;
					nErrId:=3;
				END_IF
			END_FOR
			IF  bError THEN			(*if exiest same file *)
				IF bContinueWhenErr THEN
					Step:=60;
					bError:=FALSE;
					nErrId:=0;
				ELSIF bCancelWhenErr THEN
					i:=i+1;
					bError:=FALSE;
					nErrId:=0;
				END_IF
			ELSE					(*no same file *)
				fbFileCopy
					(
					srcNetId:='' ,
					srcFileName:=CONCAT(CONCAT(CONCAT(srcPathName,DirectoryName),'\'),srcFilesLists[i].sFileName) ,
					cbReadLen:=srcFilesLists[i].fileSize.dwLowPart,
					destNetId:='' ,
					destFileName:=CONCAT(CONCAT(CONCAT(destPathName,DirectoryName),'\'),srcFilesLists[i].sFileName) ,
					bExecute:=TRUE ,
					tAdsTimeOut:=T#10s ,
					);
				Step:=60;
			END_IF
		END_IF

	60:	(*copy*)
		fbFileCopy();
		IF NOT fbFileCopy.bBusy THEN
			fbFileCopy(bExecute:=FALSE);
			IF i>=15 THEN
				i:=1;
				Step:=70;
			ELSE
				i:=i+1;
				Step:=50;
			END_IF
		END_IF

	70:	(*finish*)
		bFindFileListState:=FALSE;
		bBusy := FALSE;
		Step:=0;

END_CASE

END_FUNCTION_BLOCK

// ---- POUs/000_程序辅助系统/报警/Alarm_FB/FB_SetAlarm.TcPOU
FUNCTION_BLOCK FB_SetAlarm(*设置报警功能块,每个报警调用一次*)
VAR_INPUT
    InUse:                         	BOOL;(*是否使用*)
	EventId:						DINT;(*报警号*)
	EventMessage:                  	STRING;(*报警信息*)
	EventActive:					BOOL;(*触发信号*)
   	FilterInUse:                  	BOOL:=FALSE;(* 是否使用滤波器*)(*对触发信号进行滤波，就是触发信号超过多少时间后才报警*)
   	FilterTime:                    	TIME;(*滤波时间*)
	QuitRequired:					BOOL;(*是否自动复位: true=复位信号为1时复位报警信号;false=触发信号为0时复位报警信号*)
	QuitEvent:					 	BOOL;(*复位信号*)
	EventClass:						Alm_EventClass;(*报警等级*)
	ToTheLogFile:					BOOL;(*是否记录到历史记录文件*)
   	ToTheHistory:                 	BOOL;(*是否记录到报警历史记录*)
	(* event actions	*)
	AlarmlampOn:				BOOL;(*是否需要报警灯亮*)
	AutoRunOff:					BOOL;(*退出自动循环*)
	AlarmAction1:				BOOL;(*用户定义报警动作*)(*例如定义为黄灯亮,则该报警号有触发时,主报警程序的该输出信号为1*)
	AlarmAction2:				BOOL;(*用户定义报警动作*)
	AlarmAction3:				BOOL;(*用户定义报警动作*)
	AlarmAction4:				BOOL;(*用户定义报警动作*)
	AlarmAction5:				BOOL;(*用户定义报警动作*)
	AlarmAction6:				BOOL;(*用户定义报警动作*)
	AlarmAction7:				BOOL;(*用户定义报警动作*)
	AlarmAction8:				BOOL;(*用户定义报警动作*)	
	D1:							DINT;//
	D2:							DINT;//
	S1:							STRING(255);//
END_VAR
VAR_OUTPUT
	EventAlive:					BOOL;(*当前报警正在执行*)
  	ShowlampOn:            		BOOL;(*当前报警灯亮*)
END_VAR
VAR
 	F_Trig_QuitEvent:          	F_TRIG;
	n:                        	DINT;
	R_TRIG_GetTime:          	R_TRIG;
  	TON_Filter:               	TON;
	sTemp: 						STRING(255);//临时=wEventMessage,无时间有内容
	fbFormatStringDateTime: 	FB_FormatString;
	swFormatWstring: 			SW_FormatWstring;
	sDateTimeString: 			STRING(255);
	wEventMessage: 				WSTRING(255);//没有时间，只有信息
	wEventMessage_pre: 			WSTRING(255);//报警等级
	wmesstest							:WSTRING(255);//只有时间
	wsCurrentValue_eventclass:WSTRING(255);
END_VAR

ACT_ToTheHistory();
IF EventId> cnAlarmLast OR EventId< cnAlarmFirst THEN
	RETURN;
END_IF

(*--------------------------------------------------警报数组---------------------------------------------------*)
       (*Reset Alarm*)
	   F_Trig_QuitEvent(CLK:=QuitEvent);
       	IF (QuitRequired AND  F_Trig_QuitEvent.Q)
      	OR NOT QuitRequired AND NOT EventActive
     	OR NOT InUse THEN
              	EventAlive:=FALSE;
            	ShowlampOn:=FALSE;
				AlarmActionArray[EventId].AutoRunOff	:=FALSE;(*退出自动循环*)
             	AlarmActionArray[EventId].AlarmAction1:=FALSE;
             	AlarmActionArray[EventId].AlarmAction2:=FALSE;
            	AlarmActionArray[EventId].AlarmAction3:=FALSE;
             	AlarmActionArray[EventId].AlarmAction4:=FALSE;
             	AlarmActionArray[EventId].AlarmAction5:=FALSE;
             	AlarmActionArray[EventId].AlarmAction6:=FALSE;
            	AlarmActionArray[EventId].AlarmAction7:=FALSE;
            	AlarmActionArray[EventId].AlarmAction8:=FALSE;
				AlarmActionArray[EventId].InUse:=InUse;
				AlarmActionArray[EventId].EventAlive:=EventAlive;
				AlarmActionArray[EventId].ShowlampOn:=ShowlampOn;
				AlarmActionArray[EventId].EventActive:=EventActive;
				AlarmActionArray[EventId].EventClass:=EventClass;
				AlarmActionArray[EventId].EventId:=EventId;
				AlarmActionArray[EventId].QuitEvent:=QuitEvent;
				AlarmActionArray[EventId].QuitRequired:=QuitRequired;
       	END_IF
(*-----------------------------------------------当前激活警报数组-------------------------------------------------*)	
       (*SetAlarm*)
	 	TON_Filter(IN:=FilterInUse AND EventActive , PT:=FilterTime );
		R_TRIG_GetTime(CLK:=(NOT FilterInUse AND EventActive) OR (FilterInUse AND TON_Filter.Q)AND InUse );  
		IF R_TRIG_GetTime.Q THEN
      		AlarmActionArray[EventId].EventTime:=SYSTEMTIME_TO_DT(tActSystemTime);
		END_IF
       	IF ((NOT FilterInUse AND EventActive) OR (FilterInUse AND TON_Filter.Q)) 
		AND InUse THEN
              EventAlive:=TRUE;
              ShowlampOn:=AlarmlampOn;
              AlarmActionArray[EventId].AutoRunOff:=AutoRunOff;
              AlarmActionArray[EventId].AlarmAction1:=AlarmAction1;
              AlarmActionArray[EventId].AlarmAction2:=AlarmAction2;
              AlarmActionArray[EventId].AlarmAction3:=AlarmAction3;
              AlarmActionArray[EventId].AlarmAction4:=AlarmAction4;
              AlarmActionArray[EventId].AlarmAction5:=AlarmAction5;
              AlarmActionArray[EventId].AlarmAction6:=AlarmAction6;
              AlarmActionArray[EventId].AlarmAction7:=AlarmAction7;
              AlarmActionArray[EventId].AlarmAction8:=AlarmAction8;
			  (*I/O*)
			 AlarmActionArray[EventId].InUse:=InUse;
			 AlarmActionArray[EventId].EventAlive:=EventAlive;
			 AlarmActionArray[EventId].ShowlampOn:=ShowlampOn;
			 AlarmActionArray[EventId].EventActive:=EventActive;
			 AlarmActionArray[EventId].EventClass:=EventClass;
			 AlarmActionArray[EventId].EventId:=EventId;
			 AlarmActionArray[EventId].QuitEvent:=QuitEvent;
			 AlarmActionArray[EventId].QuitRequired:=QuitRequired;
			 
			 IF R_TRIG_GetTime.Q THEN
				 fbFormatStringDateTime(
					sFormat:= 	'%D-%D-%D-%D:%D:%D',
					arg1:= 		F_WORD(tActSystemTime.wYear),
					arg2:= 		F_WORD(tActSystemTime.wMonth),
					arg3:= 		F_WORD(tActSystemTime.wDay),
					arg4:= 		F_WORD(tActSystemTime.wHour),
					arg5:= 		F_WORD(tActSystemTime.wMinute),
					arg6:= 		F_WORD(tActSystemTime.wSecond),
					sOut=> 		sDateTimeString
					);
				//IF VisuElems.CURRENTLANGUAGE='english' THEN
					wEventMessage:=STRING_TO_WSTRING(AlarmActionArray[EventId].AlarmMsg.EN);
				//ELSE
				//	wEventMessage:=AlarmActionArray[EventId].AlarmMsg.CN;
				//END_IF
				
				(********把报警等级加入************)
				wsCurrentValue_eventclass:=TO_WSTRING(EventClass);
				wEventMessage_pre:=WCONCAT(wsCurrentValue_eventclass,":");
				
				swFormatWstring(
					WstringIn:= 	wEventMessage, 
					D1:= 			D1, 
					D2:= 			D2, 
					S1:= 			S1, 
					WstringOUT=> 	wEventMessage
					);
				
				
				//wEventMessage:=	WCONCAT(wEventMessage_pre, WCONCAT(WCONCAT(WCONCAT("ID",DINT_TO_WSTRING(EventId)),","),wEventMessage));
				wEventMessage:=	WCONCAT(wEventMessage_pre,wEventMessage);
				wmesstest := WCONCAT(STRING_TO_WSTRING(sDateTimeString),"-");	
				AlarmActionArray[EventId].EventMessage := WCONCAT(wmesstest,wEventMessage);	
			END_IF

			 
       END_IF

ACTION ACT_ToTheHistory:
(*---------------------------------------------------历史警报数组----------------------------------------------------*)
IF ToTheHistory   AND R_TRIG_GetTime.Q THEN
        Alm_HistoryAlarmNum:=Alm_HistoryAlarmNum+1;
        IF Alm_HistoryAlarmNum>=cnAlmHistoryLast THEN
               Alm_HistoryAlarmNum:=cnAlmHistoryLast;
        END_IF
        IF Alm_HistoryAlarmNum>=cnAlmHistoryFirst+1 THEN
             FOR n:=Alm_HistoryAlarmNum TO cnAlmHistoryFirst+1 BY -1 DO
                  AlarmHistoryArray[n]:=AlarmHistoryArray[n-1];
             END_FOR
        END_IF
 	AlarmHistoryArray[1].EventId:=EventId;
	AlarmHistoryArray[1].EventTime:=AlarmActionArray[EventId].EventTime;
  	AlarmHistoryArray[1].EventMessage:=AlarmActionArray[EventId].EventMessage;
END_IF
IF ToTheLogFile AND R_TRIG_GetTime.Q THEN
	wstring_to_utf8(ADR(sTemp),ADR(wEventMessage),SIZEOF(sTemp));
	gsWriteToLog:=concat(gsWriteToLog,sTemp);
END_IF
END_ACTION

END_FUNCTION_BLOCK

// ---- POUs/000_程序辅助系统/报警/MAIN_Alarm.TcPOU
PROGRAM MAIN_ALarm
VAR
	fbAlarmMAIN:						FB_AlarmMAIN;
	fbDiagDataLogging_S:				FB_DiagDataLogging_S;	
	ethercatdiag1,ethercatdiag2:		ethercatinfo_read;
	ec_alarm_trig1,ec_alarm_trig2:		Tc2_Standard.R_TRIG;
	TON_Delay: 							Ton;		
	bInidDone: 							BOOL;
	D1:									DINT:=0;//ec1 报警总数
	D2:									DINT:=0;//ec1报警模块位置
	D3:									DINT:=0;
	D4:									DINT:=0;
    D5,D6:	DINT:=0;
	ModleName1,ModleName2:				Tc2_System.T_MaxString;
	ecnumber1,ecnumber2:				DINT;
	ec_alarm1,ec_alarm2:				BOOL;
	i: 									DINT;

	a,b :INT;
	m1,m2,m3,m4:INT;
	
	Auto_clean_ton:Tc2_Standard.TON;
END_VAR

ethercatdiag_action();

IF NOT bInidDone THEN
	aInit();
ELSE
	TON_Delay(IN:=TRUE , PT:=T#2S );
	IF TON_Delay.Q THEN
		aOtherAlarm();
		fbAlarmMAIN();

		gbAlarm_StopAlarm := fbAlarmMAIN.AlarmAction1;
		gbAlarm_NeedPause := fbAlarmMAIN.AlarmAction2;
		fbDiagDataLogging_s(sInputString:=gsWriteToLog);
		
	END_IF	
END_IF

(*************定时复位历史报警***********************)
Auto_clean_ton(IN:=NOT Auto_clean_ton.Q  , PT:=T#1H , Q=> , ET=> );
IF Auto_clean_ton.Q THEN 
	Alm_bHMIClearHistory:=TRUE;
ELSE 
	Alm_bHMIClearHistory:=FALSE;
END_IF
(*报警灯*)
//GVL_IO.yelllow_lamp:=fbAlarmMAIN.FalshLamp;
(*蜂鸣*)
//GVL_IO.buzz:=fbAlarmMAIN.ShowlampOn;
(*复位*)
//Alm_bBtReset:=GVL_IO.bReast OR gvl.HMI_reset OR GVL.STOM_LBJ.reset;

ACTION aInit:
	AlarmActionArray[1].AlarmMsg.CN	:=	"ETHERCAT 1总线错误,报警数量%D,在第%D个,名称为%S";
	AlarmActionArray[2].AlarmMsg.CN	:=	"ETHERCAT 2总线错误,报警数量%D,在第%D个,名称为%S";


	AlarmActionArray[1].AlarmMsg.EN	:=	'ETHERCAT 1 error,number:%D,deviceID:%D,%S';
	AlarmActionArray[2].AlarmMsg.EN	:=	'ETHERCAT 2 error,number:%D,deviceID:%D,%S';
	AlarmActionArray[3].AlarmMsg.EN	:=	'Alarm3';
	AlarmActionArray[4].AlarmMsg.EN	:=	'Alarm4';
	AlarmActionArray[5].AlarmMsg.EN	:=	'Alarm5';
	AlarmActionArray[6].AlarmMsg.EN	:=	'Alarm6';
	AlarmActionArray[7].AlarmMsg.EN	:=	'Alarm7';
	AlarmActionArray[8].AlarmMsg.EN	:=	'Alarm8';
	AlarmActionArray[9].AlarmMsg.EN	:=	'Alarm9';

	
	
	FOR i:=cnAlarmFirst TO cnAlarmLast DO
		fbSetAlarm[i].EventId := i;
	END_FOR	
	bInidDone:=TRUE;
END_ACTION

ACTION aOtherAlarm:
ec_alarm_trig1(CLK:= ec_alarm1, Q=> );
IF ec_alarm_trig1.Q THEN
	D1:=D1+1;
END_IF
ec_alarm_trig2(CLK:= ec_alarm2, Q=> );
IF ec_alarm_trig2.Q THEN
	D3:=D3+1;
END_IF

fbSetAlarm[1](
	InUse:= TRUE, 
	EventId:= 1, 
	EventActive:= ec_alarm1, 
	QuitRequired:= , 
	QuitEvent:= , 
	EventClass:=Alm_EventClass.Alarm , 
	ToTheLogFile:= TRUE, 
	ToTheHistory:= TRUE, 
	AlarmlampOn:=  TRUE,
	AlarmAction1:= TRUE, 
	AlarmAction2:= TRUE, 
	D1:=			D1,
	D2:=			D2,
	S1:=			ModleName1,
	EventAlive=> , 
	ShowlampOn=> );
	
fbSetAlarm[2](
	InUse:= TRUE, 
	EventId:= 2, 
	EventActive:= ec_alarm2, 
	QuitRequired:= , 
	QuitEvent:= , 
	EventClass:=Alm_EventClass.Alarm ,
	ToTheLogFile:= TRUE, 
	ToTheHistory:= TRUE,
    AlarmlampOn:=  TRUE, 
	AlarmAction1:= TRUE, 
	AlarmAction2:= TRUE, 
	D1:=			D3,
	D2:=			D4,
	S1:=			ModleName2,
	EventAlive=> , 
	ShowlampOn=> );
END_ACTION

ACTION ethercatdiag_action:
ethercatdiag1(
	netID:= , 
	nEcMasterDeviceId:= , 
	slaveAddresses=> , 
	devStates=> , 
	slavenames=> , 
	color=> , 
	nSlaves=> );

IF ethercatdiag1.nSlaves >0 THEN
FOR ecnumber1 :=0 TO (ethercatdiag1.nSlaves-1)  BY 1 DO
	IF ethercatdiag1.devStates[ecnumber1].deviceState>=8 THEN
		ec_alarm1:=FALSE;
	ELSE
		ec_alarm1:=TRUE;
		D2:=ecnumber1+1;
		ModleName1:=ethercatdiag1 .slavenames[ecnumber1];
		EXIT;
	END_IF
END_FOR
END_IF

ethercatdiag2(
	netID:= , 
	nEcMasterDeviceId:= , 
	slaveAddresses=> , 
	devStates=> , 
	slavenames=> , 
	color=> , 
	nSlaves=> );

IF ethercatdiag2.nSlaves >0 THEN
FOR ecnumber2 :=0 TO (ethercatdiag2.nSlaves-1)  BY 1 DO
	IF ethercatdiag2.devStates[ecnumber2].deviceState>=8 THEN
		ec_alarm2:=FALSE;
	ELSE
		ec_alarm2:=TRUE;
		D4:=ecnumber2+1;
		ModleName2:=ethercatdiag2 .slavenames[ecnumber2];
		EXIT;
	END_IF
END_FOR
END_IF
END_ACTION

END_PROGRAM

// ---- POUs/000_程序辅助系统/系统功能/P_UPS.TcPOU
PROGRAM P_UPS
VAR
	FB_UPS: FB_S_UPS_CX51x0;                      //UPS功能块
	dataloaded: BOOL;                             //UPS数据文件读取状态(TRUE为读取成功，FALSE为读取失败)
	OldData: BOOL;                                //UPS备份数据文件读取状态
	PersistentDataStatus: EPlcPersistentStatus;   //Persistent数据读取(恢复)状态
	
   	
END_VAR

FB_UPS(
	sNetID:= ,                                //默认为本地的NetId
	iPLCPort:= ,                              //PLC运行时系统的端口号,功能块会自动获取,默认为0
	iUPSPort:= ,                              //读取PLC电源端口的状态号,默认为16#588
	tTimeout:= ,                              
	eUpsMode:= eSUPS_WrPersistData_Shutdown,  //UPS模式,即一旦保存了持久数据，就会自动执行快速关闭
	ePersistentMode:= SPDM_2PASS,             //Persistent数据的写入模式,默认为SPDM_2PASS
	tRecoverTime:= ,                          
	bPowerFailDetect=> ,                      //断电时为TRUE，如果存在电源电压，则为FALSE   
	eState=> );                               //当前UPS状态
	dataloaded:=_AppInfo.BootDataLoaded;
	OldData:=_AppInfo.OldBootData;
	PersistentDataStatus:=_AppInfo.PersistentStatus;

END_PROGRAM

// ---- POUs/001_FB/FB_count.TcPOU
FUNCTION_BLOCK FB_count
VAR_INPUT
	Add_Time:TIME;
END_VAR
VAR_OUTPUT
	count:INT;
END_VAR
VAR
	ton1:TON;
	a:INT;
END_VAR

ton1(IN:=NOT ton1.Q  , PT:=Add_Time , Q=> , ET=> );
IF ton1.Q THEN 
	count:=count+1;
END_IF
IF count>=1000 THEN 
	count:=0;
END_IF

END_FUNCTION_BLOCK

// ---- POUs/001_FB/FB_WriteAnalog.TcPOU
FUNCTION_BLOCK FB_WriteAnalog

(* 12-Bit DA-Converter for 0V~ 10V *)
(*
Measured value Decimal output Hexadecimal output
		0 V 			0 			0x0000
		5 V 			16383 		0x3FFF
		10 V 		32767 		0x7FFF
*)
VAR_INPUT
	Enable:BOOL;
	In:REAL;
	AnalogOffset:INT;
	Set_MaxValue:LREAL;
	MaxValue:REAL;
END_VAR
VAR_OUTPUT
	out:INT;
END_VAR

